(* CODESYS project CutToLength Prog final.project

Project tree, tasks and I/O mapping:
  Drive : Unidrive M701, Nidec Control Techniques, version 1.10.1.9
    application Application
      Program/
        program Freewheeling [LD]
      Codesys Setup/
        libraries: CT Unidrive M Parameter Library, * (Control Techniques); CT Unidrive M Options Parameter Library, 1.10.1.9 (Control Techniques)
        Task Configuration
          Freewheeling
      Basic AMC Library/
        03 Commands/
          Stop/
            function Stop_Motion [ST]
            function Stop_Motion_Decel [ST]
          Home/
            function Set_Position [ST]
            function Start_Homing_To_Input_4 [ST]
            function Start_Homing_To_Input_4_Then_Marker [ST]
            function Start_Homing_To_Torque [ST]
            function Start_Homing_To_Torque_Then_Input_4 [ST]
            function Start_Homing_To_Torque_Then_Marker [ST]
          Jog/
            function Start_Jog_Minus [ST]
            function Start_Jog_Plus [ST]
          Index/
            function Start_Index_ABS [ST]
            function Start_Index_INC [ST]
            function Start_Index_REF [ST]
          EGB/
            function Start_Gearing [ST]
        01 Setup/
          function AMC_Enable [ST]
          function AMC_MasterUnits [ST]
          function AMC_UserUnits [ST]
          function AMC_StopMode [ST]
        10 Other/
          function ScaleValue_DI [ST]
          function Wait_Time [ST]
        02 Feedback/
      Variables/
        AMC Variables/
          global variables gvAMC_Flags
          global variables gvAMC_Windows
          global variables gvAMC_SoftPosLimit
          global variables gvAMC_Profile
          global variables gvAMC_HardPosLimit
          global variables gvAMC_Positions
          global variables gvAMC_Cam
          global variables gvAMC_Speed
        M701 DRIVE /
          global variables gvDrive_Commands
          global variables gvDrive_Limits
          global variables gvDrive_Flags
          global variables gvDrive_Analog
          global variables gvDrive_Digital_States
          global variables gvDrive_Info
          global variables gvDrive_Keypad
          global variables gvDrive_PID1
          global variables gvDrive_PID2
          global variables gvDrive_Menu18
          global variables gvDrive_Menu19
          global variables gvDrive_Menu20
          global variables gvDrive_Digital_Inverts
        data type eMotionID
    <Empty>
    <Empty>
    <Empty>
  Advanced Link Editor
    DefaultSection
*)

// Drive/Application/Variables/eMotionID
//This enum can be used to identify the motion.

{attribute 'qualified_only'}
TYPE eMotionID :
(
	
	NA :=0,
	AbsIndex_001 		:=101,
	AbsIndex_002 		:=102,
	AbsIndex_003 		:=103,
	AbsIndex_004 		:=104,
	AbsIndex_005 		:=105,
	AbsIndex_006 		:=106,
	AbsIndex_007 		:=107,
	AbsIndex_008 		:=108,
	AbsIndex_009 		:=109,
	AbsIndex_010 		:=110, 
	
	RefIndex_001 		:=201,
	RefIndex_002 		:=202,
	RefIndex_003 		:=203,
	RefIndex_004 		:=204,
	RefIndex_005 		:=205,
	RefIndex_006 		:=206,
	RefIndex_007 		:=207,
	RefIndex_008 		:=208,
	RefIndex_009 		:=209,
	RefIndex_010 		:=210, 
	
	IncIndex_001 		:=301,
	IncIndex_002 		:=302,
	IncIndex_003 		:=303,
	IncIndex_004 		:=304,
	IncIndex_005 		:=305,
	IncIndex_006 		:=306,
	IncIndex_007 		:=307,
	IncIndex_008 		:=308,
	IncIndex_009 		:=309,
	IncIndex_010 		:=310,  

	JogPlus_001			:=401,
	JogPlus_002			:=402,
	JogPlus_003			:=403,
	JogPlus_004			:=404,
	JogPlus_005			:=405,
	JogPlus_006			:=406,
	JogPlus_007			:=407,
	JogPlus_008			:=408,
	JogPlus_009			:=409,
	JogPlus_010			:=410,

	JogMinus_001		:=501,
	JogMinus_002		:=502,
	JogMinus_003		:=503,
	JogMinus_004		:=504,
	JogMinus_005		:=505,
	JogMinus_006		:=506,
	JogMinus_007		:=507,
	JogMinus_008		:=508,
	JogMinus_009		:=509,
	JogMinus_010		:=510,

	Gearing_001			:=601,
	Gearing_002			:=602,
	Gearing_003			:=603,
	Gearing_004			:=604,
	Gearing_005			:=605,
	Gearing_006			:=606,
	Gearing_007			:=607,
	Gearing_008			:=608,
	Gearing_009			:=609,
	Gearing_010			:=610,

	Cam_001				:=701,
	Cam_002				:=702,
	Cam_003				:=703,
	Cam_004				:=704,
	Cam_005				:=705,
	Cam_006				:=706,
	Cam_007				:=707,
	Cam_008				:=708,
	Cam_009				:=709,
	Cam_010				:=710,

	Home_001			:=801,
	Home_002			:=802,
	Home_003			:=803,
	Home_004			:=804,
	Home_005			:=805,
	Home_006			:=806,
	Home_007			:=807,
	Home_008			:=808,
	Home_009			:=809,
	Home_010			:=810,
	
	
	Error	 := -1		 //
)INT;
END_TYPE

// Drive/Application/Variables/AMC Variables/gvAMC_Flags
{attribute 'qualified_only'}
VAR_GLOBAL
	
 	//(33.010) [Get:Set] AMC Slave Freeze Flag, 
	//Slave freeze flag status parameter 33.010. 
	{attribute 'get_access' := 'ReadUserParameterBOOL(00,33,010)'}
	{attribute 'set_access' := 'WriteUserParameterBOOL(00,33,010,CaptureFlag_1)'}
	{attribute 'monitoring_instead' := 'ReadUserParameterBOOL(00,33,010)'}
	CaptureFlag_1: BOOL;

	
	//(32.010) [Get:Set] AMC Master Freeze Flag, 
	//Master freeze flag status.  
	{attribute 'get_access' := 'ReadUserParameterBOOL(00,32,010)'}
	{attribute 'set_access' := 'WriteUserParameterBOOL(00,32,010,CaptureFlag_2)'}
	{attribute 'monitoring_instead' := 'ReadUserParameterBOOL(00,32,010)'}
	CaptureFlag_2: BOOL;

	
	//(37.006) AMC EGB Locked,[Get] , 
	//Displays when the electronic gearbox is locked.  
	{attribute 'get_access' := 'ReadUserParameterBOOL(00,37,006)'}
	{attribute 'monitoring_instead' := 'ReadUserParameterBOOL(00,37,006)'}
	EGB_Locked: BOOL;
	

	//(41.004) AMC Movement Complete Flag[Get] 
	//range 0 to 1 - precision is 0 decimal places.
	//NOTE:  There is a 4ms update delay for this Parameter. 
	{attribute 'get_access' := 'ReadUserParameterBOOL(00,41,004)'}
	{attribute 'monitoring_instead' := 'ReadUserParameterBOOL(00,41,004)'}
	MovementCompleteFlag: BOOL;
	
	
	//(41.004) AMC Profile Complete Flag[Get] 
	//range 0 to 1 - precision is 0 decimal places.
	//NOTE:  There is a 4ms update delay for this Parameter. 
	{attribute 'get_access' := 'ReadUserParameterBOOL(00,41,006)'}
	{attribute 'monitoring_instead' := 'ReadUserParameterBOOL(00,41,006)'}
	ProfileCompleteFlag: BOOL;
	
	
	//(40.005)[Get] Home Complete Flag 
	//Indiates that the Home is Complete.  If the Home has a offset position command the motor 
	//might not be done moving to the offset position.
	{attribute 'get_access' := 'ReadUserParameterBOOL(00,40,005)'}
	{attribute 'monitoring_instead' := 'ReadUserParameterBOOL(00,40,005)'}
	HomeCompleteFlag : BOOL;
	
		
	//(40.007)[Get] Home Complete with Offset Complete
	//Indiates that the Home and the offset move is Complete.  If the Home has a offset position command the motor 
	//might not be done moving to the offset position.
	{attribute 'get_access' := 'ReadUserParameterBOOL(00,40,008)'}
	{attribute 'monitoring_instead' := 'ReadUserParameterBOOL(00,40,008)'}
	HomeOffsetCompleteFlag : BOOL;
	 
	
	//(41.008)[Get] AMC Following Error Flag 
	//Indiates that the position error is outside the follwing error window Parameter 41.007
	{attribute 'get_access' := 'ReadUserParameterBOOL(00,41,008)'}
	{attribute 'monitoring_instead' := 'ReadUserParameterBOOL(00,41,008)'}
	FollowingErrorFlag : BOOL;
	 
	//(41.010)[Get] AMC Speed Error Flag 
	//Indiates that the position error is outside the follwing error window Parameter 41.010
	{attribute 'get_access' := 'ReadUserParameterBOOL(00,41,010)'}
	{attribute 'monitoring_instead' := 'ReadUserParameterBOOL(00,41,010)'}
	SpeedErrorFlag : BOOL;
	 
	//(41.012) [Get] AMC Following Error Stop Flag 
	{attribute 'get_access' := 'ReadUserParameterBOOL(00,41,012)'}
	{attribute 'monitoring_instead' := 'ReadUserParameterBOOL(00,41,012)'}
	FollowingErrorStop: BOOL;

	//(41.013)[Get] AMC Positive Hardware Limit Flag 
	{attribute 'get_access' := 'ReadUserParameterBOOL(00,41,013)'}
	{attribute 'monitoring_instead' := 'ReadUserParameterBOOL(00,41,013)'}
	Positive_HardwareLimit: BOOL;
	
	//(41.014) [Get] AMC Negative Hardware Limit Flag 
	{attribute 'get_access' := 'ReadUserParameterBOOL(00,41,014)'}
	{attribute 'monitoring_instead' := 'ReadUserParameterBOOL(00,41,014)'}
	Negative_HardwareLimit: BOOL;
	
	//(41.015) [Get] AMC Positive Software Limit Flag 
	{attribute 'get_access' := 'ReadUserParameterBOOL(00,41,015)'}
	{attribute 'monitoring_instead' := 'ReadUserParameterBOOL(00,41,015)'}
	Positive_SoftwareLimit: BOOL;
	
	//(41.016) [Get] AMC Negative Software Limit Flag 
	{attribute 'get_access' := 'ReadUserParameterBOOL(00,41,016)'}
	{attribute 'monitoring_instead' := 'ReadUserParameterBOOL(00,41,016)'}
	Negative_SoftwareLimit: BOOL;
	
	//(41.017)[Get] AMC Home Required Flag, 
	{attribute 'get_access' := 'ReadUserParameterBOOL(00,41,017)'}
	{attribute 'monitoring_instead' := 'ReadUserParameterBOOL(00,41,017)'}
	HomeRequired: BOOL;
	
	
	
END_VAR

// Drive/Application/Variables/AMC Variables/gvAMC_Windows
{attribute 'qualified_only'}
VAR_GLOBAL
	

	//(41.003) AMC Movement Complete Window [Get:Set] 
	// range -2147483648 to 2147483647UU - precision is 0 decimal places.
	{attribute 'get_access' 		:= 'ReadUserParameterDINT(00,41,003)'}
	{attribute 'set_access' 		:= 'WriteUserParameterDINT(00,41,003,MovementCompleteWindow)'}
	{attribute 'monitoring_instead' := 'ReadUserParameterDINT(00,41,003)'}
	MovementCompleteWindow: DINT; 

	//(41.005) AMC Profile Complete Window [Get:Set] 
	// range -2147483648 to 2147483647UU - precision is 0 decimal places.
	{attribute 'get_access' 		:= 'ReadUserParameterDINT(00,41,005)'}
	{attribute 'set_access' 		:= 'WriteUserParameterDINT(00,41,005,ProfileCompleteWindow)'}
	{attribute 'monitoring_instead' := 'ReadUserParameterDINT(00,41,005)'}
	ProfileCompleteWindow: DINT; 

	//(41.007) AMC Following Error Window [Get:Set] 
	// range -2147483648 to 2147483647UU - precision is 0 decimal places.
	{attribute 'get_access' 		:= 'ReadUserParameterDINT(00,41,007)'}
	{attribute 'set_access' 		:= 'WriteUserParameterDINT(00,41,007,FollowingErrorWindow)'}
	{attribute 'monitoring_instead' := 'ReadUserParameterDINT(00,41,007)'}
	FollowingErrorWindow: DINT; 

	//(41.009) AMC At Speed Window [Get:Set] 
	// range -2147483648 to 2147483647UU - precision is 0 decimal places.
	{attribute 'get_access' 		:= 'ReadUserParameterDINT(00,41,009)'}
	{attribute 'set_access' 		:= 'WriteUserParameterDINT(00,41,009,AtSpeedWindow)'}
	{attribute 'monitoring_instead' := 'ReadUserParameterDINT(00,41,009)'}
	AtSpeedWindow: DINT; 
	
	
	
END_VAR

// Drive/Application/Variables/AMC Variables/gvAMC_SoftPosLimit
{attribute 'qualified_only'}
VAR_GLOBAL
  
	
 	//(41.024) AMC Enable Software Limits, [Get:Set], 
	//range 0 to 1   
	//Value of 0 = Profile
	//Value of 1 = No Profile
	{attribute 'get_access' 		:= 'ReadUserParameterSINT (00,41,024)'}
	{attribute 'set_access' 		:= 'WriteUserParameterSINT(00,41,024,SoftwareLimitStopMode)'}
	{attribute 'monitoring_instead' := 'ReadUserParameterSINT (00,41,024)'}
	SoftwareLimitStopMode		: SINT;
	 
  	//(41.025) AMC Enable Software Limits, [Get:Set], 
	//range 0 to 1   
	{attribute 'get_access' 		:= 'ReadUserParameterBOOL (00,41,025)'}
	{attribute 'set_access' 		:= 'WriteUserParameterBOOL(00,41,025,EnableSoftwareLimits)'}
	{attribute 'monitoring_instead' := 'ReadUserParameterBOOL (00,41,025)'}
	EnableSoftwareLimits		: BOOL;	 
	
	//(41.026)AMC Positive Software Limit Position, [Get:Set] , 
	//range -2147483648 to 2147483647UU - precision is 0 decimal places. 
	{attribute 'get_access' 		:= 'ReadUserParameterDINT  (00,41,026)'}
	{attribute 'set_access' 		:= 'WriteUserParameterDINT (00,41,026,PositiveSoftwareLimitPosition)'}
	{attribute 'monitoring_instead' := 'ReadUserParameterDINT  (00,41,026)'}
	PositiveSoftwareLimitPosition: DINT;
	
	
	//(41.027) AMC Negative Software Limit Position, [Get:Set] , 
	//range -2147483648 to 2147483647UU - precision is 0 decimal places. 
	{attribute 'get_access' 		:= 'ReadUserParameterDINT (00,41,027)'}
	{attribute 'set_access' 		:= 'WriteUserParameterDINT(00,41,027,NegativeSoftwareLimitPosition)'}
	{attribute 'monitoring_instead' := 'ReadUserParameterDINT (00,41,027)'}
	NegativeSoftwareLimitPosition: DINT;
	
	
	
END_VAR

// Drive/Application/Variables/AMC Variables/gvAMC_Profile
{attribute 'qualified_only'}
VAR_GLOBAL
	
  
	
	//(38.001) [Get:Set] AMC Profile Acceleration, range -2147483648 to 2147483647UU/ms²
	// precision is 3 decimal places.
	// Unit are in User units / ms² 
	{attribute 'get_access' 		:= 'ReadUserParameterDINT(00,38,001)'}
	{attribute 'set_access' 		:= 'WriteUserParameterDINT(00,38,001,Acceleration)'}
	{attribute 'monitoring_instead' := 'ReadUserParameterDINT(00,38,001)'}
	Acceleration: DINT; 
	
	//(38.002) [Get:Set] AMC Profile Deceleration, range -2147483648 to 2147483647UU/ms²
	// precision is 3 decimal places.
	// Unit are in User units / ms² 
	{attribute 'get_access' 		:= 'ReadUserParameterDINT(00,38,002)'}
	{attribute 'set_access' 		:= 'WriteUserParameterDINT(00,38,002,Deceleration)'}
	{attribute 'monitoring_instead' := 'ReadUserParameterDINT(00,38,002)'}
	Deceleration: DINT; 
	
	//(38.003) [Get:Set] AMC Profile Maximum Speed, range -2147483648 to 2147483647UU/ms
	//precision is 2 decimal places.
	//Unit are in User units / ms
	{attribute 'get_access' 		:= 'ReadUserParameterDINT(00,38,003)'}
	{attribute 'set_access' 		:= 'WriteUserParameterDINT(00,38,003,MaximumSpeed)'}
	{attribute 'monitoring_instead' := 'ReadUserParameterDINT(00,38,003)'}
	MaximumSpeed: DINT;
	
	
END_VAR

// Drive/Application/Variables/AMC Variables/gvAMC_HardPosLimit
{attribute 'qualified_only'}
VAR_GLOBAL
	 

	//(41.023) AMC Hardware Limit Stop Mode, [Get:Set]  
	//Stop mode used when a hardware limit are active. 
	//Value of 0 = Profile
	//Value of 1 = No Profile
	//This uses parameter 6.035 and parameter 6.036.
	//parameter 06.035 is Forward Limit Switch 
	//parameter 06.036 is Reverse Limit Switch
	//These two parameters are controled by anything you map to it.  Most of the time a digital input will control them.
	//Example:  Set parameter 8.025 = 6.035 and set parameter 8.026 = 6.036.  Now digital input 5 and 6 control the hardware limits.
	{attribute 'get_access' 		:= 'ReadUserParameterSINT(00,41,023)'}
	{attribute 'set_access' 		:= 'WriteUserParameterSINT(00,41,023,HardwareLimitSwitch_NoRamp_StopMode)'}
	{attribute 'monitoring_instead' := 'ReadUserParameterSINT(00,41,023)'}	
	HardwareLimitSwitch_NoRamp_StopMode			: SINT;
 
   
	 
	 
	
END_VAR

// Drive/Application/Variables/AMC Variables/gvAMC_Positions
{attribute 'qualified_only'}
VAR_GLOBAL
	 

	//(33.004) [Get] System Position, range -2147483648 to 2147483647UU - 
	//precision is 0 decimal places.
	//Displays the AMC Slave Position. 
	//Update Rate 4ms
	{attribute 'get_access' 		:= 'ReadUserParameterDINT(00,33,004)'}
	{attribute 'monitoring_instead' := 'ReadUserParameterDINT(00,33,004)'}
	SystemPosition: DINT;
  
  	//(32.004) [Get] Master Position, range -2147483648 to 2147483647UU -
	//precision is 0 decimal places. 
	//Displays the AMC Slave Position. 
	//Update Rate 4ms
	{attribute 'get_access' 		:= 'ReadUserParameterDINT(00,32,004)'}
	{attribute 'monitoring_instead' := 'ReadUserParameterDINT(00,32,004)'}
	MasterPosition: DINT; 
	
	 
	//[Get] AMC Slave Freeze Position(33.006),  
	//Displays the AMC Slave Position after a freeze event has occurred. 
	{attribute 'get_access' 		:= 'ReadUserParameterDINT(00,33,006)'}
	{attribute 'monitoring_instead' := 'ReadUserParameterDINT(00,33,006)'}
	CapturedPosition_1: DINT;
	
	
	///[Get] AMC Master Freeze Position(32.006), 
	//Displays the AMC Slave Position after a freeze event has occurred. 
	{attribute 'get_access' 		:= 'ReadUserParameterDINT(00,32,006)'}
	{attribute 'monitoring_instead' := 'ReadUserParameterDINT(00,32,006)'}
	CapturedPosition_2: DINT;
	
	
END_VAR

// Drive/Application/Variables/M701 DRIVE /gvDrive_Commands
{attribute 'qualified_only'}
VAR_GLOBAL
	 

	//(06.008)Hold Zero Speed [Get:Set] 
	//If True then the drive will hold a zero speed command even if no run command is given
	{attribute 'get_access' 		:= 'ReadUserParameterBOOL (00,06,008)'}
	{attribute 'set_access' 		:= 'WriteUserParameterBOOL(00,06,008,HoldZeroSpeed)'}
	{attribute 'monitoring_instead' := 'ReadUserParameterBOOL (00,06,008)'}
	HoldZeroSpeed : BOOL;

	
	//(06.030) Basic Run Forward [Get:Set] 
	//Needs to be true before anymoon commands will operate.
	{attribute 'get_access' 		:= 'ReadUserParameterBOOL (00,06,030)'}
	{attribute 'set_access' 		:= 'WriteUserParameterBOOL(00,06,030,RunForward)'}
	{attribute 'monitoring_instead' := 'ReadUserParameterBOOL (00,06,030)'}
	RunForward: BOOL;
	
	 
	//(06.032) Basic Run Reverse [Get:Set] 
	//Needs to be true before anymoon commands will operate.
	{attribute 'get_access' 		:= 'ReadUserParameterBOOL (00,06,032)'}
	{attribute 'set_access' 		:= 'WriteUserParameterBOOL(00,06,032,RunReverse)'}
	{attribute 'monitoring_instead' := 'ReadUserParameterBOOL (00,06,032)'}
	RunReverse: BOOL;
	
	
	
END_VAR

// Drive/Application/Variables/M701 DRIVE /gvDrive_Limits
{attribute 'qualified_only'}
VAR_GLOBAL
	

 
	//(04.005) Motoring Current Limit [Get:Set], range 0.0 to 1000.0%
	//Defines the current limit used when the motor is being accelerated away from standstill. 
	{attribute 'get_access' 		:= 'ReadUserParameterINT (00,04,005)'}
	{attribute 'set_access' 		:= 'WriteUserParameterINT(00,04,005,MotorCurrentLimit_RAW)'}
	{attribute 'monitoring_instead' := 'ReadUserParameterINT (00,04,005)'}
	MotorCurrentLimit_RAW: INT;
 
	
	//(04.006) Regenerating Current Limit [Get:Set], range 0.0 to 1000.0%
	//Defines the current limit used when the motor is being decelerated towards standstill. 
	{attribute 'get_access' 		:= 'ReadUserParameterINT (00,04,006)'}
	{attribute 'set_access' 		:= 'WriteUserParameterINT(00,04,006,RegCurrentLimit_RAW)'}
	{attribute 'monitoring_instead' := 'ReadUserParameterINT (00,04,006)'}
	RegCurrentLimit_RAW: INT;  
	
 
	//(03.008) Over Speed Threshold, range 0.0 to 3000.0Hz
	//Set to the required over speed threshold. 
	{attribute 'get_access' 		:= 'ReadUserParameterUINT(00,03,008)'}
	{attribute 'set_access'	 		:= 'WriteUserParameterUINT(00,03,008,OverSpeedThreshold_RAW)'}
	{attribute 'monitoring_instead' := 'ReadUserParameterUINT(00,03,008)'}
	OverSpeedThreshold_RAW: UINT; 
	
	
	//(01.006) Maximum Reference Clamp [Get:Set], range -2147483648 to 2147483647 - precision is 1 decimal places.
	//Defines the maximum value for the reference. 
	{attribute 'get_access' 		:= 'ReadUserParameterDINT(00,01,006)'}
	{attribute 'set_access' 		:= 'WriteUserParameterDINT(00,01,006,MaximumReferenceClamp_RAW)'}
	{attribute 'monitoring_instead' := 'ReadUserParameterDINT(00,01,006)'}
	MaximumReferenceClamp_RAW: DINT; 
	
	
	//(01.007) Minimum Reference Clamp [Get:Set], range -2147483648 to 2147483647 - precision is 1 decimal places.
	//Defines the minimum value for the reference.  
	{attribute 'get_access' 		:= 'ReadUserParameterDINT(00,01,007)'}
	{attribute 'set_access' 		:= 'WriteUserParameterDINT(00,01,007,MinimumReferenceClamp_RAW)'}
	{attribute 'monitoring_instead' := 'ReadUserParameterDINT(00,01,007)'}
	MinimumReferenceClamp_RAW: DINT;

	
END_VAR

// Drive/Application/Variables/M701 DRIVE /gvDrive_Flags
{attribute 'qualified_only'}
VAR_GLOBAL
	
	//(10.001)[Get] Drive Healthy,  
	//Indicates that the drive is healthy. 
	{attribute 'get_access' 		:= 'ReadUserParameterBOOL(00,10,001)'}
	{attribute 'monitoring_instead' := 'ReadUserParameterBOOL(00,10,001)'}
	DriveHealthy: BOOL;
	
	//(10.003)[Get] Zero Speed,  
	//Indicates that the speed is below the zero speed threshold. 
	//Zero Speed is set to TRUE, IF the Speed Feedback parameter (03.002) 
	//is AT OR below Zero Speed Threshold (03.005).  
	{attribute 'get_access' 		:= 'ReadUserParameterBOOL(00,10,003)'}
	{attribute 'monitoring_instead' := 'ReadUserParameterBOOL(00,10,003)'}
	ZeroSpeed: BOOL;
	
	//(10.006)[Get] At Speed 
	//Indicates that the drive is running at the set speed.  
	//At Speed (10.006) is set if the Speed Feedback (03.002) is on the boundaries or 
	//within the at speed window. Above Set Speed (10.007) and Below Set Speed (10.005) 
	//are set if the feedback is above or below the window respectively.
	{attribute 'get_access' 		:= 'ReadUserParameterBOOL(00,10,006)'}
	{attribute 'monitoring_instead' := 'ReadUserParameterBOOL(00,10,006)'}
	AtSpeed : BOOL;
	
	//(10.009)[Get] Current Limit Active,  
	//Indicates that the current limit is active.  
	//is set to one if the current limit is active. 
	//It should be noted that the current limit system is used in RFC-A and RFC-S modes 
	//when standard ramp control is active (Ramp Mode (02.004)), or supply loss control 
	//is in ramp stop or limit stop mode (Supply Loss Mode (06.003)). 
	//Therefore Current Limit Active (10.009) is likely to change to one under these 
	//conditions, even if the user defined current limits are not active.
	{attribute 'get_access' 		:= 'ReadUserParameterBOOL(00,10,009)'}
	{attribute 'monitoring_instead' := 'ReadUserParameterBOOL(00,10,009)'}
	CurrentLimitActive: BOOL;

  	//(10.014)[Get] Reverse Direction Running 
	//Indicates that the drive is running in the reverse direction.  
	//Is set to one if the Speed Feedback (03.002) is negative otherwise it is set to zero. 
	{attribute 'get_access' 		:= 'ReadUserParameterBOOL(00,10,014)'}
	{attribute 'monitoring_instead' := 'ReadUserParameterBOOL(00,10,014)'}
	ReverseDirectionRunning : BOOL;
	
	
END_VAR

// Drive/Application/Variables/M701 DRIVE /gvDrive_Analog
{attribute 'qualified_only'}
VAR_GLOBAL
	
	// 07.001
   	// Analog Input 1(07.001), range -100.00-100.00
    {attribute 'get_access' 		:= 'ReadUserParameterINT(00,07,001)'}
    {attribute 'monitoring_instead' := 'ReadUserParameterINT(00,07,001)'}
    Input1_RAW : INT; 

	// 07.002
    // Analog Input 2(07.002), range -100.00-100.00.
    {attribute 'get_access' 		:= 'ReadUserParameterINT(00,07,002)'}
    {attribute 'monitoring_instead' := 'ReadUserParameterINT(00,07,002)'}
    Input2_RAW : INT;


	// 07.003
    // Analog Input 3(07.003), range -100.00-100.00.
    {attribute 'get_access' 		:= 'ReadUserParameterINT(00,07,003)'}
    {attribute 'monitoring_instead' := 'ReadUserParameterINT(00,07,003)'}
    Input3_RAW : INT;



END_VAR

// Drive/Application/Variables/M701 DRIVE /gvDrive_Digital_States
(*
	If you change the name of the inverts in this list you also have to change the set_access line of code.
	
*)

{attribute 'qualified_only'}
VAR_GLOBAL
	
	// M08.P001
    // Digital I/O 01 State
    {attribute 'get_access' 		:= 'ReadUserParameterBOOL(00,08,001)'}
    {attribute 'monitoring_instead' := 'ReadUserParameterBOOL(00,08,001)'}
    IO_01 : BOOL;

	// M08.P002	
    // Digital I/O 02 State 
    {attribute 'get_access' 		:= 'ReadUserParameterBOOL(00,08,002)'}
    {attribute 'monitoring_instead' := 'ReadUserParameterBOOL(00,08,002)'}
    IO_02 : BOOL;

	// M08.P003
    // Digital I/O 03 State 
    {attribute 'get_access' 		:= 'ReadUserParameterBOOL(00,08,003)'}
    {attribute 'monitoring_instead' := 'ReadUserParameterBOOL(00,08,003)'}
    IO_03: BOOL;

	// M08.P004
    // Digital Input 04 State 
    {attribute 'get_access' 		:= 'ReadUserParameterBOOL(00,08,004)'}
    {attribute 'monitoring_instead' := 'ReadUserParameterBOOL(00,08,004)'}
    Input04 : BOOL;
	
	// M08.P005
    // Digital Input 05 State
    {attribute 'get_access' 		:= 'ReadUserParameterBOOL(00,08,005)'}
    {attribute 'monitoring_instead' := 'ReadUserParameterBOOL(00,08,005)'}
    Input05: BOOL;

	// M08.P006
    // Digital Input 06 State
    {attribute 'get_access' 		:= 'ReadUserParameterBOOL(00,08,006)'}
    {attribute 'monitoring_instead' := 'ReadUserParameterBOOL(00,08,006)'}
    Input06 : BOOL;
 
	// M08.P007
    // Relay Output State 
    {attribute 'get_access' 		:= 'ReadUserParameterBOOL(00,08,007)'}
    {attribute 'monitoring_instead' := 'ReadUserParameterBOOL(00,08,007)'}
    RelayOutput07 : BOOL;

	// M08.P008
    // 24V Supply Output State 
    {attribute 'get_access' 		:= 'ReadUserParameterBOOL(00,08,008)'}
    {attribute 'monitoring_instead' := 'ReadUserParameterBOOL(00,08,008)'}
    VoltageSupplyOutputState  		: BOOL;

	// M08.P043
    // 24V Supply Input State 
	// Turns on when the drive is given 24v from a power supply 
    {attribute 'get_access' 		:= 'ReadUserParameterBOOL(00,08,008)'}
    {attribute 'monitoring_instead' := 'ReadUserParameterBOOL(00,08,008)'}
    VoltageSupplyInputState  		: BOOL;

	// M08.P009
    // STO Input 01 State
    {attribute 'get_access' 		:= 'ReadUserParameterBOOL(00,08,009)'}
    {attribute 'monitoring_instead' := 'ReadUserParameterBOOL(00,08,009)'}
    SaftTorqueOff1 : BOOL;

	// M08.P040	
	// STO Input 02 State 
    {attribute 'get_access' 		:= 'ReadUserParameterBOOL(00,08,040)'}
    {attribute 'monitoring_instead' := 'ReadUserParameterBOOL(00,08,040)'}
    SaftTorqueOff2 : BOOL;

END_VAR

// Drive/Application/Variables/M701 DRIVE /gvDrive_Info
{attribute 'qualified_only'}
VAR_GLOBAL
	

	//(03.002) Speed Feedback, 1 decimal places.
	//Displays the speed feedback from the selected feedback source. 
	{attribute 'get_access' 		:= 'ReadUserParameterLREAL(00,03,002)'}
	{attribute 'monitoring_instead' := 'ReadUserParameterLREAL(00,03,002)'}
	SpeedFeedback: LREAL;
	
	//(03.002) Speed Feedback, 1 decimal place, Value of 1000 = 100.0 RPM
	///Displays the speed feedback from the selected feedback source. 
	{attribute 'get_access' 		:= 'ReadUserParameterDINT(00,03,002)'}
	{attribute 'monitoring_instead' := 'ReadUserParameterDINT(00,03,002)'}
	SpeedFeedback_RAW: DINT;	
	
	//(04.001) Current Magnitude, 3 decimal places.
	//Shows the instantaneous drive output current.  
	{attribute 'get_access' 		:= 'ReadUserParameterLREAL(00,04,001)'}
	{attribute 'monitoring_instead' := 'ReadUserParameterLREAL(00,04,001)'}
	CurrentMagnitude: LREAL;	
	
	//(04.001) Current Magnitude, 3 decimal places, Value of 1000 = 1.000amps
	//Shows the instantaneous drive output current.  
	{attribute 'get_access' 		:= 'ReadUserParameterDINT(00,04,001)'}
	{attribute 'monitoring_instead' := 'ReadUserParameterDINT(00,04,001)'}
	CurrentMagnitude_RAW: DINT;	
	
	//(06.043) Control Word Enable,  
	//Set to 1 to enable the control word. - All Modes
	//if on then the control word is used to give the drive run commands
	{attribute 'get_access' 		:= 'ReadUserParameterBOOL(00,06,043)'} 
	{attribute 'set_access' 		:= 'WriteUserParameterBOOL(00,06,043,ControlWordEnable)'}
	{attribute 'monitoring_instead' := 'ReadUserParameterBOOL(00,06,043)'}
	ControlWordEnable: BOOL;
	
END_VAR

// Drive/Application/Variables/M701 DRIVE /gvDrive_Keypad
{attribute 'qualified_only'}
VAR_GLOBAL
	
 
	// M08.P041	Run Button
    {attribute 'get_access' 		:= 'ReadUserParameterBOOL(00,08,041)'}
    {attribute 'monitoring_instead' := 'ReadUserParameterBOOL(00,08,041)'}
    RunButton : BOOL;

	// M08.P042	Auxiliary Button
    {attribute 'get_access' 		:= 'ReadUserParameterBOOL(00,08,042)'}
    {attribute 'monitoring_instead' := 'ReadUserParameterBOOL(00,08,042)'}
    AuxiliaryButton : BOOL;

	// M08.P044	Auxiliary Button
    {attribute 'get_access' 		:= 'ReadUserParameterBOOL(00,08,044)'}
    {attribute 'monitoring_instead' := 'ReadUserParameterBOOL(00,08,044)'}
    StopButton : BOOL;


END_VAR

// Drive/Application/Variables/M701 DRIVE /gvDrive_PID1
(*
	See menu 14 for all of th PID settings.
*)
{attribute 'qualified_only'}
VAR_GLOBAL
		
	//(14.008) [Get:Set] PID1 Enable, 
	//Enables the use of PID1
	//Note there are also two other parameters they can be used to encable the PID
	//Parameter 14.009 and parameter 14.027
	{attribute 'get_access' 		:= 'ReadUserParameterBOOL(00,14,008)'}
	{attribute 'set_access' 		:= 'WriteUserParameterBOOL(00,14,008,Enable)'}
	{attribute 'monitoring_instead' := 'ReadUserParameterBOOL(00,14,008)'}
	Enable: BOOL;
	
	//(14.001) [Get] PID1 Output, range -100.00 to 100.00%
	//Displays the output for PID1. 
	{abvibute 'get_access' 			:= 'ReadUserParameterINT(00,14,001)'}
	{attribute 'monitoring_instead' := 'ReadUserParameterINT(00,14,001)'}
	Output_RAW: INT;

	//(14.007) [Get:Set] PID1 Reference Slew Rate, range 0.0 to 3200.0s
	//Defines the rate in change of output for PID1. 
	{attribute 'get_access' 		:= 'ReadUserParameterINT(00,14,007)'}
	{attribute 'set_access' 		:= 'WriteUserParameterINT(00,14,007,SlewRate_RAW)'}
	{attribute 'monitoring_instead' := 'ReadUserParameterINT(00,14,007)'}
	SlewRate_RAW: INT;
 
	//(14.025) [Get:Set] PID1 Digital Reference, range -100.00 to 100.00%
	//Defines the value of the digital reference for PID1. 
	//Used if the PLC is setting the Reference else the parameter 14.003 should be used.
	{attribute 'get_access' 		:= 'ReadUserParameterINT(00,14,025)'}
	{attribute 'set_access' 		:= 'WriteUserParameterINT(00,14,025,Reference_RAW)'}
	{attribute 'monitoring_instead' := 'ReadUserParameterINT(00,14,025)'}
	Reference_RAW: INT;

	//(14.026) [Get:Set] PID1 Digital Feedback, range -100.00 to 100.00%
	//Defines the value of the digital feedback for PID1. 
	//Usd if the PLC is setting the Feedback else the parameter 14.004 should be used.
	{attribute 'get_access' 		:= 'ReadUserParameterINT(00,14,026)'}
	{attribute 'set_access' 		:= 'WriteUserParameterINT(00,14,026,Feedback_RAW)'}
	{attribute 'monitoring_instead' := 'ReadUserParameterINT(00,14,026)'}
	Feedback_RAW: INT;
END_VAR

// Drive/Application/Variables/M701 DRIVE /gvDrive_PID2
(*
	See menu 14 for all of th PID settings.
*)
{attribute 'qualified_only'}
VAR_GLOBAL
	
	//(14.038) [Get:Set] PID2 Enable, 
	//Enables the use of PID2
	//Note there are also two other parameters they can be used to encable the PID
	//Parameter 14.039 and parameter 14.057
	{attribute 'get_access' 		:= 'ReadUserParameterBOOL(00,14,038)'}
	{attribute 'set_access' 		:= 'WriteUserParameterBOOL(00,14,038,Enable)'}
	{attribute 'monitoring_instead' := 'ReadUserParameterBOOL(00,14,038)'}
	Enable: BOOL;

	//(14.031) [Get] PID2 Output, range -100.00 to 100.00%
	//Displays the output for PID1. 
	{attribute 'get_access' 		:= 'ReadUserParameterINT(00,14,031)'}
	{attribute 'monitoring_instead' := 'ReadUserParameterINT(00,14,031)'}
	Output_RAW: INT;

	//(14.037) [Get:Set] PID2 Reference Slew Rate, range 0.0 to 3200.0s
	//Defines the rate in change of output for PID1. 
	{attribute 'get_access' 		:= 'ReadUserParameterINT(00,14,037)'}
	{attribute 'set_access' 		:= 'WriteUserParameterINT(00,14,037,SlewRate_RAW)'}
	{attribute 'monitoring_instead' := 'ReadUserParameterINT(00,14,037)'}
	SlewRate_RAW: INT;
 
	//(14.055) [Get:Set] PID2 Digital Reference, range -100.00 to 100.00%
	//Defines the value of the digital reference for PID1. 
	//Used if the PLC is setting the Reference else the parameter 14.003 should be used.
	{attribute 'get_access' 		:= 'ReadUserParameterINT(00,14,055)'}
	{attribute 'set_access' 		:= 'WriteUserParameterINT(00,14,055,Reference_RAW)'}
	{attribute 'monitoring_instead' := 'ReadUserParameterINT(00,14,055)'}
	Reference_RAW: INT;

	//(14.056) [Get:Set] PID2 Digital Feedback, range -100.00 to 100.00%
	//Defines the value of the digital feedback for PID1. 
	//Usd if the PLC is setting the Feedback else the parameter 14.004 should be used.
	{attribute 'get_access' 		:= 'ReadUserParameterINT(00,14,056)'}
	{attribute 'set_access' 		:= 'WriteUserParameterINT(00,14,056,Feedback_RAW)'}
	{attribute 'monitoring_instead' := 'ReadUserParameterINT(00,14,056)'}
	Feedback_RAW: INT;
END_VAR

// Drive/Application/Variables/M701 DRIVE /gvDrive_Menu18
(*
	Menu 18
*)
(*	LEVEL 2 SUPPORT
	Only change the variable name after you know how.
	don't add extra white spaces inside the attribute.
*)
(*
	If you change the name of any of them in this list you also have to change the set_access line of code.
	
	Example:
	change P001 to P001_count
	Then you also need to change the attributes
 
	before
	
	{attribute 'get_bitaccess' := 'ReadUserParameterBit(00,18,001,BITNR)'}
	{attribute 'get_access' := 'ReadUserParameterINT(00,18,001)'}
	{attribute 'set_bitaccess' := 'WriteUserParameterBit(00,18,001,BITNR,P001)'}
	{attribute 'set_access' := 'WriteUserParameterINT(00,18,001,P001)'}
	{attribute 'monitoring_instead' := 'ReadUserParameterINT(00,18,001)'}
	P001: INT;
	
	after change 
	
	{attribute 'get_bitaccess' := 'ReadUserParameterBit(00,18,001,BITNR)'}
	{attribute 'get_access' := 'ReadUserParameterINT(00,18,001)'}
	{attribute 'set_bitaccess' := 'WriteUserParameterBit(00,18,001,BITNR,P001_count)'}
	{attribute 'set_access' := 'WriteUserParameterINT(00,18,001,P001_count)'}
	{attribute 'monitoring_instead' := 'ReadUserParameterINT(00,18,001)'}
	P001_count: INT;
	
*)
{attribute 'qualified_only'}
VAR_GLOBAL
 
	
	//(18.001)
	//save on power down
	{attribute 'get_bitaccess' := 'ReadUserParameterBit(00,18,001,BITNR)'}
	{attribute 'get_access' := 'ReadUserParameterINT(00,18,001)'}
	{attribute 'set_bitaccess' := 'WriteUserParameterBit(00,18,001,BITNR,Length_mm)'}
	{attribute 'set_access' := 'WriteUserParameterINT(00,18,001,Length_mm)'}
	{attribute 'monitoring_instead' := 'ReadUserParameterINT(00,18,001)'}
	Length_mm: INT;
	
	//(18.002) 
	{attribute 'get_bitaccess' := 'ReadUserParameterBit(00,18,002,BITNR)'}
	{attribute 'get_access' := 'ReadUserParameterINT(00,18,002)'}
	{attribute 'set_bitaccess' := 'WriteUserParameterBit(00,18,002,BITNR,View_Speed_Percent)'}
	{attribute 'set_access' := 'WriteUserParameterINT(00,18,002,View_Speed_Percent)'}
	{attribute 'monitoring_instead' := 'ReadUserParameterINT(00,18,002)'}
	View_Speed_Percent: INT;
	
	// (18.003) 
	{attribute 'get_bitaccess' := 'ReadUserParameterBit(00,18,003,BITNR)'}
	{attribute 'get_access' := 'ReadUserParameterINT(00,18,003)'}
	{attribute 'set_bitaccess' := 'WriteUserParameterBit(00,18,003,BITNR,Drive_Status)'}
	{attribute 'set_access' := 'WriteUserParameterINT(00,18,003,Drive_Status)'}
	{attribute 'monitoring_instead' := 'ReadUserParameterINT(00,18,003)'}
	Drive_Status: INT;
	
	//(18.004) 
	{attribute 'get_bitaccess' := 'ReadUserParameterBit(00,18,004,BITNR)'}
	{attribute 'get_access' := 'ReadUserParameterINT(00,18,004)'}
	{attribute 'set_bitaccess' := 'WriteUserParameterBit(00,18,004,BITNR,Count_Display)'}
	{attribute 'set_access' := 'WriteUserParameterINT(00,18,004,Count_Display)'}
	{attribute 'monitoring_instead' := 'ReadUserParameterINT(00,18,004)'}
	Count_Display: INT;
	
	//(18.005) 
	{attribute 'get_bitaccess' := 'ReadUserParameterBit(00,18,005,BITNR)'}
	{attribute 'get_access' := 'ReadUserParameterINT(00,18,005)'}
	{attribute 'set_bitaccess' := 'WriteUserParameterBit(00,18,005,BITNR,View_Distance_Per_Motor_Turn)'}
	{attribute 'set_access' := 'WriteUserParameterINT(00,18,005,View_Distance_Per_Motor_Turn)'}
	{attribute 'monitoring_instead' := 'ReadUserParameterINT(00,18,005)'}
	View_Distance_Per_Motor_Turn: INT;
	
	//(18.006) 
	{attribute 'get_bitaccess' := 'ReadUserParameterBit(00,18,006,BITNR)'}
	{attribute 'get_access' := 'ReadUserParameterINT(00,18,006)'}
	{attribute 'set_bitaccess' := 'WriteUserParameterBit(00,18,006,BITNR,View_Distance_Per_Encoder_Turn)'}
	{attribute 'set_access' := 'WriteUserParameterINT(00,18,006,View_Distance_Per_Encoder_Turn)'}
	{attribute 'monitoring_instead' := 'ReadUserParameterINT(00,18,006)'}
	View_Distance_Per_Encoder_Turn: INT;
	
	//(18.007) 
	{attribute 'get_bitaccess' := 'ReadUserParameterBit(00,18,007,BITNR)'}
	{attribute 'get_access' := 'ReadUserParameterINT(00,18,007)'}
	{attribute 'set_bitaccess' := 'WriteUserParameterBit(00,18,007,BITNR,View_Acceleration_Position)'}
	{attribute 'set_access' := 'WriteUserParameterINT(00,18,007,View_Acceleration_Position)'}
	{attribute 'monitoring_instead' := 'ReadUserParameterINT(00,18,007)'}
	View_Acceleration_Position: INT;
	
	//(18.008)
	{attribute 'get_bitaccess' := 'ReadUserParameterBit(00,18,008,BITNR)'}
	{attribute 'get_access' := 'ReadUserParameterINT(00,18,008)'}
	{attribute 'set_bitaccess' := 'WriteUserParameterBit(00,18,008,BITNR,View_Decceleration_Position)'}
	{attribute 'set_access' := 'WriteUserParameterINT(00,18,008,View_Decceleration_Position)'}
	{attribute 'monitoring_instead' := 'ReadUserParameterINT(00,18,008)'}
	View_Decceleration_Position: INT;
	
	//(18.009)
	{attribute 'get_bitaccess' := 'ReadUserParameterBit(00,18,009,BITNR)'}
	{attribute 'get_access' := 'ReadUserParameterINT(00,18,009)'}
	{attribute 'set_bitaccess' := 'WriteUserParameterBit(00,18,009,BITNR,View_Jog_Acceleration)'}
	{attribute 'set_access' := 'WriteUserParameterINT(00,18,009,View_Jog_Acceleration)'}
	{attribute 'monitoring_instead' := 'ReadUserParameterINT(00,18,009)'}
	View_Jog_Acceleration: INT;
	
	//(18.010) 
	{attribute 'get_bitaccess' := 'ReadUserParameterBit(00,18,010,BITNR)'}
	{attribute 'get_access' := 'ReadUserParameterINT(00,18,010)'}
	{attribute 'set_bitaccess' := 'WriteUserParameterBit(00,18,010,BITNR,View_Jog_Decceleration)'}
	{attribute 'set_access' := 'WriteUserParameterINT(00,18,010,View_Jog_Decceleration)'}
	{attribute 'monitoring_instead' := 'ReadUserParameterINT(00,18,010)'}
	View_Jog_Decceleration: INT;
	
	//(18.011) 
	{attribute 'get_bitaccess' := 'ReadUserParameterBit(00,18,011,BITNR)'}
	{attribute 'get_access' := 'ReadUserParameterINT(00,18,011)'}
	{attribute 'set_bitaccess' := 'WriteUserParameterBit(00,18,011,BITNR,View_Jog_Speed)'}
	{attribute 'set_access' := 'WriteUserParameterINT(00,18,011,View_Jog_Speed)'}
	{attribute 'monitoring_instead' := 'ReadUserParameterINT(00,18,011)'}
	View_Jog_Speed: INT;
	
	//(18.012) 
	{attribute 'get_bitaccess' := 'ReadUserParameterBit(00,18,012,BITNR)'}
	{attribute 'get_access' := 'ReadUserParameterINT(00,18,012)'}
	{attribute 'set_bitaccess' := 'WriteUserParameterBit(00,18,012,BITNR,Speed_Percent)'}
	{attribute 'set_access' := 'WriteUserParameterINT(00,18,012,Speed_Percent)'}
	{attribute 'monitoring_instead' := 'ReadUserParameterINT(00,18,012)'}
	Speed_Percent: INT := 150;
	
	//(18.013) 
	{attribute 'get_bitaccess' := 'ReadUserParameterBit(00,18,013,BITNR)'}
	{attribute 'get_access' := 'ReadUserParameterINT(00,18,013)'}
	{attribute 'set_bitaccess' := 'WriteUserParameterBit(00,18,013,BITNR,Count_Preset)'}
	{attribute 'set_access' := 'WriteUserParameterINT(00,18,013,Count_Preset)'}
	{attribute 'monitoring_instead' := 'ReadUserParameterINT(00,18,013)'}
	Count_Preset: INT := 0;
	
	//(18.014) 
	{attribute 'get_bitaccess' := 'ReadUserParameterBit(00,18,014,BITNR)'}
	{attribute 'get_access' := 'ReadUserParameterINT(00,18,014)'}
	{attribute 'set_bitaccess' := 'WriteUserParameterBit(00,18,014,BITNR,P014)'}
	{attribute 'set_access' := 'WriteUserParameterINT(00,18,014,P014)'}
	{attribute 'monitoring_instead' := 'ReadUserParameterINT(00,18,014)'}
	P014: INT;
	
	//(18.015)
	{attribute 'get_bitaccess' := 'ReadUserParameterBit(00,18,015,BITNR)'}
	{attribute 'get_access' := 'ReadUserParameterINT(00,18,015)'}
	{attribute 'set_bitaccess' := 'WriteUserParameterBit(00,18,015,BITNR,P015)'}
	{attribute 'set_access' := 'WriteUserParameterINT(00,18,015,P015)'}
	{attribute 'monitoring_instead' := 'ReadUserParameterINT(00,18,015)'}
	P015: INT;
	
	//(18.016)
	{attribute 'get_bitaccess' := 'ReadUserParameterBit(00,18,016,BITNR)'}
	{attribute 'get_access' := 'ReadUserParameterINT(00,18,016)'}
	{attribute 'set_bitaccess' := 'WriteUserParameterBit(00,18,016,BITNR,P016)'}
	{attribute 'set_access' := 'WriteUserParameterINT(00,18,016,P016)'}
	{attribute 'monitoring_instead' := 'ReadUserParameterINT(00,18,016)'}
	P016: INT;
	
	//(18.017)
	{attribute 'get_bitaccess' := 'ReadUserParameterBit(00,18,017,BITNR)'}
	{attribute 'get_access' := 'ReadUserParameterINT(00,18,017)'}
	{attribute 'set_bitaccess' := 'WriteUserParameterBit(00,18,017,BITNR,P017)'}
	{attribute 'set_access' := 'WriteUserParameterINT(00,18,017,P017)'}
	{attribute 'monitoring_instead' := 'ReadUserParameterINT(00,18,017)'}
	P017: INT;
	
	//(18.018)
	{attribute 'get_bitaccess' := 'ReadUserParameterBit(00,18,018,BITNR)'}
	{attribute 'get_access' := 'ReadUserParameterINT(00,18,018)'}
	{attribute 'set_bitaccess' := 'WriteUserParameterBit(00,18,018,BITNR,P018)'}
	{attribute 'set_access' := 'WriteUserParameterINT(00,18,018,P018)'}
	{attribute 'monitoring_instead' := 'ReadUserParameterINT(00,18,018)'}
	P018: INT;
	
	//(18.019) 
	{attribute 'get_bitaccess' := 'ReadUserParameterBit(00,18,019,BITNR)'}
	{attribute 'get_access' := 'ReadUserParameterINT(00,18,019)'}
	{attribute 'set_bitaccess' := 'WriteUserParameterBit(00,18,019,BITNR,P019)'}
	{attribute 'set_access' := 'WriteUserParameterINT(00,18,019,P019)'}
	{attribute 'monitoring_instead' := 'ReadUserParameterINT(00,18,019)'}
	P019: INT;
	
	//(18.020)
	{attribute 'get_bitaccess' := 'ReadUserParameterBit(00,18,020,BITNR)'}
	{attribute 'get_access' := 'ReadUserParameterINT(00,18,020)'}
	{attribute 'set_bitaccess' := 'WriteUserParameterBit(00,18,020,BITNR,P020)'}
	{attribute 'set_access' := 'WriteUserParameterINT(00,18,020,P020)'}
	{attribute 'monitoring_instead' := 'ReadUserParameterINT(00,18,020)'}
	P020: INT;
	
	//(18.021)
	{attribute 'get_bitaccess' := 'ReadUserParameterBit(00,18,021,BITNR)'}
	{attribute 'get_access' := 'ReadUserParameterINT(00,18,021)'}
	{attribute 'set_bitaccess' := 'WriteUserParameterBit(00,18,021,BITNR,P021)'}
	{attribute 'set_access' := 'WriteUserParameterINT(00,18,021,P021)'}
	{attribute 'monitoring_instead' := 'ReadUserParameterINT(00,18,021)'}
	P021: INT;
	
	//(18.022) 
	{attribute 'get_bitaccess' := 'ReadUserParameterBit(00,18,022,BITNR)'}
	{attribute 'get_access' := 'ReadUserParameterINT(00,18,022)'}
	{attribute 'set_bitaccess' := 'WriteUserParameterBit(00,18,022,BITNR,P022)'}
	{attribute 'set_access' := 'WriteUserParameterINT(00,18,022,P022)'}
	{attribute 'monitoring_instead' := 'ReadUserParameterINT(00,18,022)'}
	P022: INT;
	
	//(18.023) 
	{attribute 'get_bitaccess' := 'ReadUserParameterBit(00,18,023,BITNR)'}
	{attribute 'get_access' := 'ReadUserParameterINT(00,18,023)'}
	{attribute 'set_bitaccess' := 'WriteUserParameterBit(00,18,023,BITNR,P023)'}
	{attribute 'set_access' := 'WriteUserParameterINT(00,18,023,P023)'}
	{attribute 'monitoring_instead' := 'ReadUserParameterINT(00,18,023)'}
	P023: INT;
	
	//(18.024) 
	{attribute 'get_bitaccess' := 'ReadUserParameterBit(00,18,024,BITNR)'}
	{attribute 'get_access' := 'ReadUserParameterINT(00,18,024)'}
	{attribute 'set_bitaccess' := 'WriteUserParameterBit(00,18,024,BITNR,P024)'}
	{attribute 'set_access' := 'WriteUserParameterINT(00,18,024,P024)'}
	{attribute 'monitoring_instead' := 'ReadUserParameterINT(00,18,024)'}
	P024: INT;
	
	//(18.025)
	{attribute 'get_bitaccess' := 'ReadUserParameterBit(00,18,025,BITNR)'}
	{attribute 'get_access' := 'ReadUserParameterINT(00,18,025)'}
	{attribute 'set_bitaccess' := 'WriteUserParameterBit(00,18,025,BITNR,P025)'}
	{attribute 'set_access' := 'WriteUserParameterINT(00,18,025,P025)'}
	{attribute 'monitoring_instead' := 'ReadUserParameterINT(00,18,025)'}
	P025: INT;
	
	//(18.026)
	{attribute 'get_bitaccess' := 'ReadUserParameterBit(00,18,026,BITNR)'}
	{attribute 'get_access' := 'ReadUserParameterINT(00,18,026)'}
	{attribute 'set_bitaccess' := 'WriteUserParameterBit(00,18,026,BITNR,P026)'}
	{attribute 'set_access' := 'WriteUserParameterINT(00,18,026,P026)'}
	{attribute 'monitoring_instead' := 'ReadUserParameterINT(00,18,026)'}
	P026: INT;
	
	//(18.027)
	{attribute 'get_bitaccess' := 'ReadUserParameterBit(00,18,027,BITNR)'}
	{attribute 'get_access' := 'ReadUserParameterINT(00,18,027)'}
	{attribute 'set_bitaccess' := 'WriteUserParameterBit(00,18,027,BITNR,P027)'}
	{attribute 'set_access' := 'WriteUserParameterINT(00,18,027,P027)'}
	{attribute 'monitoring_instead' := 'ReadUserParameterINT(00,18,027)'}
	P027: INT;
	
	//(18.028)
	{attribute 'get_bitaccess' := 'ReadUserParameterBit(00,18,028,BITNR)'}
	{attribute 'get_access' := 'ReadUserParameterINT(00,18,028)'}
	{attribute 'set_bitaccess' := 'WriteUserParameterBit(00,18,028,BITNR,P028)'}
	{attribute 'set_access' := 'WriteUserParameterINT(00,18,028,P028)'}
	{attribute 'monitoring_instead' := 'ReadUserParameterINT(00,18,028)'}
	P028: INT;
	
	//(18.029)
	{attribute 'get_bitaccess' := 'ReadUserParameterBit(00,18,029,BITNR)'}
	{attribute 'get_access' := 'ReadUserParameterINT(00,18,029)'}
	{attribute 'set_bitaccess' := 'WriteUserParameterBit(00,18,029,BITNR,P029)'}
	{attribute 'set_access' := 'WriteUserParameterINT(00,18,029,P029)'}
	{attribute 'monitoring_instead' := 'ReadUserParameterINT(00,18,029)'}
	P029: INT;
	
	//(18.030)
	{attribute 'get_bitaccess' := 'ReadUserParameterBit(00,18,030,BITNR)'}
	{attribute 'get_access' := 'ReadUserParameterINT(00,18,030)'}
	{attribute 'set_bitaccess' := 'WriteUserParameterBit(00,18,030,BITNR,P030)'}
	{attribute 'set_access' := 'WriteUserParameterINT(00,18,030,P030)'}
	{attribute 'monitoring_instead' := 'ReadUserParameterINT(00,18,030)'}
	P030: INT;
	
	//(18.031) 
	{attribute 'get_access' := 'ReadUserParameterBOOL(00,18,031)'} 
	{attribute 'set_access' := 'WriteUserParameterBOOL(00,18,031,P031)'}
	{attribute 'monitoring_instead' := 'ReadUserParameterBOOL(00,18,031)'}
	P031: BOOL;
	
	//(18.032) 
	{attribute 'get_access' := 'ReadUserParameterBOOL(00,18,032)'} 
	{attribute 'set_access' := 'WriteUserParameterBOOL(00,18,032,P032)'}
	{attribute 'monitoring_instead' := 'ReadUserParameterBOOL(00,18,032)'}
	P032: BOOL;
	
	//(18.033) 
	{attribute 'get_access' := 'ReadUserParameterBOOL(00,18,033)'} 
	{attribute 'set_access' := 'WriteUserParameterBOOL(00,18,033,P033)'}
	{attribute 'monitoring_instead' := 'ReadUserParameterBOOL(00,18,033)'}
	P033: BOOL;
	
	//(18.034) 
	{attribute 'get_access' := 'ReadUserParameterBOOL(00,18,034)'} 
	{attribute 'set_access' := 'WriteUserParameterBOOL(00,18,034,P034)'}
	{attribute 'monitoring_instead' := 'ReadUserParameterBOOL(00,18,034)'}
	P034: BOOL;
	
	//(18.035) 
	{attribute 'get_access' := 'ReadUserParameterBOOL(00,18,035)'} 
	{attribute 'set_access' := 'WriteUserParameterBOOL(00,18,035,P035)'}
	{attribute 'monitoring_instead' := 'ReadUserParameterBOOL(00,18,035)'}
	P035: BOOL;
	
	//(18.036) 
	{attribute 'get_access' := 'ReadUserParameterBOOL(00,18,036)'} 
	{attribute 'set_access' := 'WriteUserParameterBOOL(00,18,036,P036)'}
	{attribute 'monitoring_instead' := 'ReadUserParameterBOOL(00,18,036)'}
	P036: BOOL;
	
	//(18.037)  
	{attribute 'get_access' := 'ReadUserParameterBOOL(00,18,037)'} 
	{attribute 'set_access' := 'WriteUserParameterBOOL(00,18,037,P037)'}
	{attribute 'monitoring_instead' := 'ReadUserParameterBOOL(00,18,037)'}
	P037: BOOL;
	
	//(18.038)  
	{attribute 'get_access' := 'ReadUserParameterBOOL(00,18,038)'} 
	{attribute 'set_access' := 'WriteUserParameterBOOL(00,18,038,P038)'}
	{attribute 'monitoring_instead' := 'ReadUserParameterBOOL(00,18,038)'}
	P038: BOOL;
	
	//(18.039)
	{attribute 'get_access' := 'ReadUserParameterBOOL(00,18,039)'} 
	{attribute 'set_access' := 'WriteUserParameterBOOL(00,18,039,P039)'}
	{attribute 'monitoring_instead' := 'ReadUserParameterBOOL(00,18,039)'}
	P039: BOOL;
	
	//(18.040)
	{attribute 'get_access' := 'ReadUserParameterBOOL(00,18,040)'} 
	{attribute 'set_access' := 'WriteUserParameterBOOL(00,18,040,P040)'}
	{attribute 'monitoring_instead' := 'ReadUserParameterBOOL(00,18,040)'}
	P040: BOOL;
	
	//(18.041) 
	{attribute 'get_access' := 'ReadUserParameterBOOL(00,18,041)'} 
	{attribute 'set_access' := 'WriteUserParameterBOOL(00,18,041,P041)'}
	{attribute 'monitoring_instead' := 'ReadUserParameterBOOL(00,18,041)'}
	P041: BOOL;
	
	//(18.042) 
	{attribute 'get_access' := 'ReadUserParameterBOOL(00,18,042)'} 
	{attribute 'set_access' := 'WriteUserParameterBOOL(00,18,042,P042)'}
	{attribute 'monitoring_instead' := 'ReadUserParameterBOOL(00,18,042)'}
	P042: BOOL;
	
	//(18.043) 
	{attribute 'get_access' := 'ReadUserParameterBOOL(00,18,043)'} 
	{attribute 'set_access' := 'WriteUserParameterBOOL(00,18,043,P043)'}
	{attribute 'monitoring_instead' := 'ReadUserParameterBOOL(00,18,043)'}
	P043: BOOL;
	
	//(18.044) 
	{attribute 'get_access' := 'ReadUserParameterBOOL(00,18,044)'} 
	{attribute 'set_access' := 'WriteUserParameterBOOL(00,18,044,P044)'}
	{attribute 'monitoring_instead' := 'ReadUserParameterBOOL(00,18,044)'}
	P044: BOOL;
	
	//18.045) 
	{attribute 'get_access' := 'ReadUserParameterBOOL(00,18,045)'} 
	{attribute 'set_access' := 'WriteUserParameterBOOL(00,18,045,P045)'}
	{attribute 'monitoring_instead' := 'ReadUserParameterBOOL(00,18,045)'}
	P045: BOOL;
	
	//(18.046) 
	{attribute 'get_access' := 'ReadUserParameterBOOL(00,18,046)'} 
	{attribute 'set_access' := 'WriteUserParameterBOOL(00,18,046,P046)'}
	{attribute 'monitoring_instead' := 'ReadUserParameterBOOL(00,18,046)'}
	P046: BOOL;
	
	//(18.047) 
	{attribute 'get_access' := 'ReadUserParameterBOOL(00,18,047)'} 
	{attribute 'set_access' := 'WriteUserParameterBOOL(00,18,047,P047)'}
	{attribute 'monitoring_instead' := 'ReadUserParameterBOOL(00,18,047)'}
	P047: BOOL;
	
	//(18.048)  
	{attribute 'get_access' := 'ReadUserParameterBOOL(00,18,048)'} 
	{attribute 'set_access' := 'WriteUserParameterBOOL(00,18,048,P048)'}
	{attribute 'monitoring_instead' := 'ReadUserParameterBOOL(00,18,048)'}
	P048: BOOL;
	
	//(18.049) 
	{attribute 'get_access' := 'ReadUserParameterBOOL(00,18,049)'} 
	{attribute 'set_access' := 'WriteUserParameterBOOL(00,18,049,P049)'}
	{attribute 'monitoring_instead' := 'ReadUserParameterBOOL(00,18,049)'}
	P049: BOOL;
	
	//(18.050)  
	{attribute 'get_access' := 'ReadUserParameterBOOL(00,18,050)'} 
	{attribute 'set_access' := 'WriteUserParameterBOOL(00,18,050,P050)'}
	{attribute 'monitoring_instead' := 'ReadUserParameterBOOL(00,18,050)'}
	P050: BOOL;
	
	//(18.051) 
	{attribute 'get_bitaccess' := 'ReadUserParameterBit(00,18,051,BITNR)'}
	{attribute 'get_access' := 'ReadUserParameterDINT(00,18,051)'}
	{attribute 'set_bitaccess' := 'WriteUserParameterBit(00,18,051,BITNR,Distance_Per_Motor_Turn)'}
	{attribute 'set_access' := 'WriteUserParameterDINT(00,18,051,Distance_Per_Motor_Turn)'}
	{attribute 'monitoring_instead' := 'ReadUserParameterDINT(00,18,051)'}
	Distance_Per_Motor_Turn: DINT := 25;
	
	//(18.052) 
	{attribute 'get_bitaccess' := 'ReadUserParameterBit(00,18,052,BITNR)'}
	{attribute 'get_access' := 'ReadUserParameterDINT(00,18,052)'}
	{attribute 'set_bitaccess' := 'WriteUserParameterBit(00,18,052,BITNR,Distance_Per_Encoder_Turn)'}
	{attribute 'set_access' := 'WriteUserParameterDINT(00,18,052,Distance_Per_Encoder_Turn)'}
	{attribute 'monitoring_instead' := 'ReadUserParameterDINT(00,18,052)'}
	Distance_Per_Encoder_Turn: DINT := 360;
	
	//18.053) 
	{attribute 'get_bitaccess' := 'ReadUserParameterBit(00,18,053,BITNR)'}
	{attribute 'get_access' := 'ReadUserParameterDINT(00,18,053)'}
	{attribute 'set_bitaccess' := 'WriteUserParameterBit(00,18,053,BITNR,Acceleration_Position)'}
	{attribute 'set_access' := 'WriteUserParameterDINT(00,18,053,Acceleration_Position)'}
	{attribute 'monitoring_instead' := 'ReadUserParameterDINT(00,18,053)'}
	Acceleration_Position: DINT := 100;
	

	//(18.054) 
	{attribute 'get_bitaccess' := 'ReadUserParameterBit(00,18,054,BITNR)'}
	{attribute 'get_access' := 'ReadUserParameterDINT(00,18,054)'}
	{attribute 'set_bitaccess' := 'WriteUserParameterBit(00,18,054,BITNR,Decceleration_Position)'}
	{attribute 'set_access' := 'WriteUserParameterDINT(00,18,054,Decceleration_Position)'}
	{attribute 'monitoring_instead' := 'ReadUserParameterDINT(00,18,054)'}
	Decceleration_Position: DINT := 100;
	
END_VAR

// Drive/Application/Variables/AMC Variables/gvAMC_Cam
{attribute 'qualified_only'}
VAR_GLOBAL
	  
	//(35.007) Displays which index in the Cam table the Cam controller is using
	//Update Rate 4ms
	{attribute 'get_access' := 'ReadUserParameterINT(00,35,007)'}
	{attribute 'monitoring_instead' := 'ReadUserParameterINT(00,35,007)'}
	Segment_Index: INT;
  
	//(35.008) Displays the position in the segment that the cam controller is using
	//Update Rate 4ms
	{attribute 'get_access' := 'ReadUserParameterDINT(00,35,008)'}
	{attribute 'monitoring_instead' := 'ReadUserParameterDINT(00,35,008)'}
	Position_In_Segment: DINT;
 
	//(35.010) Displays when the cam controller reaches the end of the cam table
	//Update Rate 4ms
	{attribute 'get_access' := 'ReadUserParameterBOOL(00,35,010)'}
	{attribute 'monitoring_instead' := 'ReadUserParameterBOOL(00,35,010)'}
	Cam_Complete: BOOL;
	 
END_VAR

// Drive/Application/Variables/M701 DRIVE /gvDrive_Menu19
(*
	Menu 19
*)
(*	LEVEL 2 SUPPORT
	Only change the variable name after you know how.
	don't add extra white spaces inside the attribute.
*)
(*
	If you change the name of any of them in this list you also have to change the set_access line of code.
	
	Example:
	change P001 to P001_count
	Then you also need to change the attributes
 
	before
	
	{attribute 'get_bitaccess' := 'ReadUserParameterBit(00,19,001,BITNR)'}
	{attribute 'get_access' := 'ReadUserParameterINT(00,19,001)'}
	{attribute 'set_bitaccess' := 'WriteUserParameterBit(00,19,001,BITNR,P001)'}
	{attribute 'set_access' := 'WriteUserParameterINT(00,19,001,P001)'}
	{attribute 'monitoring_instead' := 'ReadUserParameterINT(00,19,001)'}
	P001: INT;
	
	after change 
	
	{attribute 'get_bitaccess' := 'ReadUserParameterBit(00,19,001,BITNR)'}
	{attribute 'get_access' := 'ReadUserParameterINT(00,19,001)'}
	{attribute 'set_bitaccess' := 'WriteUserParameterBit(00,19,001,BITNR,P001_count)'}
	{attribute 'set_access' := 'WriteUserParameterINT(00,19,001,P001_count)'}
	{attribute 'monitoring_instead' := 'ReadUserParameterINT(00,19,001)'}
	P001_count: INT;
	
*)
{attribute 'qualified_only'}
VAR_GLOBAL
 
	
	//(19.001)
	//save on power down
	{attribute 'get_bitaccess' := 'ReadUserParameterBit(00,19,001,BITNR)'}
	{attribute 'get_access' := 'ReadUserParameterINT(00,19,001)'}
	{attribute 'set_bitaccess' := 'WriteUserParameterBit(00,19,001,BITNR,P001)'}
	{attribute 'set_access' := 'WriteUserParameterINT(00,19,001,P001)'}
	{attribute 'monitoring_instead' := 'ReadUserParameterINT(00,19,001)'}
	P001: INT;
	
	//(19.002) 
	{attribute 'get_bitaccess' := 'ReadUserParameterBit(00,19,002,BITNR)'}
	{attribute 'get_access' := 'ReadUserParameterINT(00,19,002)'}
	{attribute 'set_bitaccess' := 'WriteUserParameterBit(00,19,002,BITNR,P002)'}
	{attribute 'set_access' := 'WriteUserParameterINT(00,19,002,P002)'}
	{attribute 'monitoring_instead' := 'ReadUserParameterINT(00,19,002)'}
	P002: INT;
	
	// (19.003) 
	{attribute 'get_bitaccess' := 'ReadUserParameterBit(00,19,003,BITNR)'}
	{attribute 'get_access' := 'ReadUserParameterINT(00,19,003)'}
	{attribute 'set_bitaccess' := 'WriteUserParameterBit(00,19,003,BITNR,P003)'}
	{attribute 'set_access' := 'WriteUserParameterINT(00,19,003,P003)'}
	{attribute 'monitoring_instead' := 'ReadUserParameterINT(00,19,003)'}
	P003: INT;
	
	//(19.004) 
	{attribute 'get_bitaccess' := 'ReadUserParameterBit(00,19,004,BITNR)'}
	{attribute 'get_access' := 'ReadUserParameterINT(00,19,004)'}
	{attribute 'set_bitaccess' := 'WriteUserParameterBit(00,19,004,BITNR,P004)'}
	{attribute 'set_access' := 'WriteUserParameterINT(00,19,004,P004)'}
	{attribute 'monitoring_instead' := 'ReadUserParameterINT(00,19,004)'}
	P004: INT;
	
	//(19.005) 
	{attribute 'get_bitaccess' := 'ReadUserParameterBit(00,19,005,BITNR)'}
	{attribute 'get_access' := 'ReadUserParameterINT(00,19,005)'}
	{attribute 'set_bitaccess' := 'WriteUserParameterBit(00,19,005,BITNR,P005)'}
	{attribute 'set_access' := 'WriteUserParameterINT(00,19,005,P005)'}
	{attribute 'monitoring_instead' := 'ReadUserParameterINT(00,19,005)'}
	P005: INT;
	
	//(19.006) 
	{attribute 'get_bitaccess' := 'ReadUserParameterBit(00,19,006,BITNR)'}
	{attribute 'get_access' := 'ReadUserParameterINT(00,19,006)'}
	{attribute 'set_bitaccess' := 'WriteUserParameterBit(00,19,006,BITNR,P006)'}
	{attribute 'set_access' := 'WriteUserParameterINT(00,19,006,P006)'}
	{attribute 'monitoring_instead' := 'ReadUserParameterINT(00,19,006)'}
	P006: INT;
	
	//(19.007) 
	{attribute 'get_bitaccess' := 'ReadUserParameterBit(00,19,007,BITNR)'}
	{attribute 'get_access' := 'ReadUserParameterINT(00,19,007)'}
	{attribute 'set_bitaccess' := 'WriteUserParameterBit(00,19,007,BITNR,P007)'}
	{attribute 'set_access' := 'WriteUserParameterINT(00,19,007,P007)'}
	{attribute 'monitoring_instead' := 'ReadUserParameterINT(00,19,007)'}
	P007: INT;
	
	//(19.008)
	{attribute 'get_bitaccess' := 'ReadUserParameterBit(00,19,008,BITNR)'}
	{attribute 'get_access' := 'ReadUserParameterINT(00,19,008)'}
	{attribute 'set_bitaccess' := 'WriteUserParameterBit(00,19,008,BITNR,P008)'}
	{attribute 'set_access' := 'WriteUserParameterINT(00,19,008,P008)'}
	{attribute 'monitoring_instead' := 'ReadUserParameterINT(00,19,008)'}
	P008: INT;
	
	//(19.009)
	{attribute 'get_bitaccess' := 'ReadUserParameterBit(00,19,009,BITNR)'}
	{attribute 'get_access' := 'ReadUserParameterINT(00,19,009)'}
	{attribute 'set_bitaccess' := 'WriteUserParameterBit(00,19,009,BITNR,P009)'}
	{attribute 'set_access' := 'WriteUserParameterINT(00,19,009,P009)'}
	{attribute 'monitoring_instead' := 'ReadUserParameterINT(00,19,009)'}
	P009: INT;
	
	//(19.010) 
	{attribute 'get_bitaccess' := 'ReadUserParameterBit(00,19,010,BITNR)'}
	{attribute 'get_access' := 'ReadUserParameterINT(00,19,010)'}
	{attribute 'set_bitaccess' := 'WriteUserParameterBit(00,19,010,BITNR,P010)'}
	{attribute 'set_access' := 'WriteUserParameterINT(00,19,010,P010)'}
	{attribute 'monitoring_instead' := 'ReadUserParameterINT(00,19,010)'}
	P010: INT;
	
	//(19.011) 
	{attribute 'get_bitaccess' := 'ReadUserParameterBit(00,19,011,BITNR)'}
	{attribute 'get_access' := 'ReadUserParameterINT(00,19,011)'}
	{attribute 'set_bitaccess' := 'WriteUserParameterBit(00,19,011,BITNR,P011)'}
	{attribute 'set_access' := 'WriteUserParameterINT(00,19,011,P011)'}
	{attribute 'monitoring_instead' := 'ReadUserParameterINT(00,19,011)'}
	P011: INT;
	
	//(19.012) 
	{attribute 'get_bitaccess' := 'ReadUserParameterBit(00,19,012,BITNR)'}
	{attribute 'get_access' := 'ReadUserParameterINT(00,19,012)'}
	{attribute 'set_bitaccess' := 'WriteUserParameterBit(00,19,012,BITNR,P012)'}
	{attribute 'set_access' := 'WriteUserParameterINT(00,19,012,P012)'}
	{attribute 'monitoring_instead' := 'ReadUserParameterINT(00,19,012)'}
	P012: INT;
	
	//(19.013) 
	{attribute 'get_bitaccess' := 'ReadUserParameterBit(00,19,013,BITNR)'}
	{attribute 'get_access' := 'ReadUserParameterINT(00,19,013)'}
	{attribute 'set_bitaccess' := 'WriteUserParameterBit(00,19,013,BITNR,P013)'}
	{attribute 'set_access' := 'WriteUserParameterINT(00,19,013,P013)'}
	{attribute 'monitoring_instead' := 'ReadUserParameterINT(00,19,013)'}
	P013: INT;
	
	//(19.014) 
	{attribute 'get_bitaccess' := 'ReadUserParameterBit(00,19,014,BITNR)'}
	{attribute 'get_access' := 'ReadUserParameterINT(00,19,014)'}
	{attribute 'set_bitaccess' := 'WriteUserParameterBit(00,19,014,BITNR,P014)'}
	{attribute 'set_access' := 'WriteUserParameterINT(00,19,014,P014)'}
	{attribute 'monitoring_instead' := 'ReadUserParameterINT(00,19,014)'}
	P014: INT;
	
	//(19.015)
	{attribute 'get_bitaccess' := 'ReadUserParameterBit(00,19,015,BITNR)'}
	{attribute 'get_access' := 'ReadUserParameterINT(00,19,015)'}
	{attribute 'set_bitaccess' := 'WriteUserParameterBit(00,19,015,BITNR,P015)'}
	{attribute 'set_access' := 'WriteUserParameterINT(00,19,015,P015)'}
	{attribute 'monitoring_instead' := 'ReadUserParameterINT(00,19,015)'}
	P015: INT;
	
	//(19.016)
	{attribute 'get_bitaccess' := 'ReadUserParameterBit(00,19,016,BITNR)'}
	{attribute 'get_access' := 'ReadUserParameterINT(00,19,016)'}
	{attribute 'set_bitaccess' := 'WriteUserParameterBit(00,19,016,BITNR,P016)'}
	{attribute 'set_access' := 'WriteUserParameterINT(00,19,016,P016)'}
	{attribute 'monitoring_instead' := 'ReadUserParameterINT(00,19,016)'}
	P016: INT;
	
	//(19.017)
	{attribute 'get_bitaccess' := 'ReadUserParameterBit(00,19,017,BITNR)'}
	{attribute 'get_access' := 'ReadUserParameterINT(00,19,017)'}
	{attribute 'set_bitaccess' := 'WriteUserParameterBit(00,19,017,BITNR,P017)'}
	{attribute 'set_access' := 'WriteUserParameterINT(00,19,017,P017)'}
	{attribute 'monitoring_instead' := 'ReadUserParameterINT(00,19,017)'}
	P017: INT;
	
	//(19.018)
	{attribute 'get_bitaccess' := 'ReadUserParameterBit(00,19,018,BITNR)'}
	{attribute 'get_access' := 'ReadUserParameterINT(00,19,018)'}
	{attribute 'set_bitaccess' := 'WriteUserParameterBit(00,19,018,BITNR,P018)'}
	{attribute 'set_access' := 'WriteUserParameterINT(00,19,019,P018)'}
	{attribute 'monitoring_instead' := 'ReadUserParameterINT(00,19,018)'}
	P018: INT;
	
	//(19.019) 
	{attribute 'get_bitaccess' := 'ReadUserParameterBit(00,19,019,BITNR)'}
	{attribute 'get_access' := 'ReadUserParameterINT(00,19,019)'}
	{attribute 'set_bitaccess' := 'WriteUserParameterBit(00,19,019,BITNR,P019)'}
	{attribute 'set_access' := 'WriteUserParameterINT(00,19,019,P019)'}
	{attribute 'monitoring_instead' := 'ReadUserParameterINT(00,19,019)'}
	P019: INT;
	
	//(19.020)
	{attribute 'get_bitaccess' := 'ReadUserParameterBit(00,19,020,BITNR)'}
	{attribute 'get_access' := 'ReadUserParameterINT(00,19,020)'}
	{attribute 'set_bitaccess' := 'WriteUserParameterBit(00,19,020,BITNR,P020)'}
	{attribute 'set_access' := 'WriteUserParameterINT(00,19,020,P020)'}
	{attribute 'monitoring_instead' := 'ReadUserParameterINT(00,19,020)'}
	P020: INT;
	
	//(19.021)
	{attribute 'get_bitaccess' := 'ReadUserParameterBit(00,19,021,BITNR)'}
	{attribute 'get_access' := 'ReadUserParameterINT(00,19,021)'}
	{attribute 'set_bitaccess' := 'WriteUserParameterBit(00,19,021,BITNR,P021)'}
	{attribute 'set_access' := 'WriteUserParameterINT(00,19,021,P021)'}
	{attribute 'monitoring_instead' := 'ReadUserParameterINT(00,19,021)'}
	P021: INT;
	
	//(19.022) 
	{attribute 'get_bitaccess' := 'ReadUserParameterBit(00,19,022,BITNR)'}
	{attribute 'get_access' := 'ReadUserParameterINT(00,19,022)'}
	{attribute 'set_bitaccess' := 'WriteUserParameterBit(00,19,022,BITNR,P022)'}
	{attribute 'set_access' := 'WriteUserParameterINT(00,19,022,P022)'}
	{attribute 'monitoring_instead' := 'ReadUserParameterINT(00,19,022)'}
	P022: INT;
	
	//(19.023) 
	{attribute 'get_bitaccess' := 'ReadUserParameterBit(00,19,023,BITNR)'}
	{attribute 'get_access' := 'ReadUserParameterINT(00,19,023)'}
	{attribute 'set_bitaccess' := 'WriteUserParameterBit(00,19,023,BITNR,P023)'}
	{attribute 'set_access' := 'WriteUserParameterINT(00,19,023,P023)'}
	{attribute 'monitoring_instead' := 'ReadUserParameterINT(00,19,023)'}
	P023: INT;
	
	//(19.024) 
	{attribute 'get_bitaccess' := 'ReadUserParameterBit(00,19,024,BITNR)'}
	{attribute 'get_access' := 'ReadUserParameterINT(00,19,024)'}
	{attribute 'set_bitaccess' := 'WriteUserParameterBit(00,19,024,BITNR,P024)'}
	{attribute 'set_access' := 'WriteUserParameterINT(00,19,024,P024)'}
	{attribute 'monitoring_instead' := 'ReadUserParameterINT(00,19,024)'}
	P024: INT;
	
	//(19.025)
	{attribute 'get_bitaccess' := 'ReadUserParameterBit(00,19,025,BITNR)'}
	{attribute 'get_access' := 'ReadUserParameterINT(00,19,025)'}
	{attribute 'set_bitaccess' := 'WriteUserParameterBit(00,19,025,BITNR,P025)'}
	{attribute 'set_access' := 'WriteUserParameterINT(00,19,025,P025)'}
	{attribute 'monitoring_instead' := 'ReadUserParameterINT(00,19,025)'}
	P025: INT;
	
	//(19.026)
	{attribute 'get_bitaccess' := 'ReadUserParameterBit(00,19,026,BITNR)'}
	{attribute 'get_access' := 'ReadUserParameterINT(00,19,026)'}
	{attribute 'set_bitaccess' := 'WriteUserParameterBit(00,19,026,BITNR,P026)'}
	{attribute 'set_access' := 'WriteUserParameterINT(00,19,026,P026)'}
	{attribute 'monitoring_instead' := 'ReadUserParameterINT(00,19,026)'}
	P026: INT;
	
	//(19.027)
	{attribute 'get_bitaccess' := 'ReadUserParameterBit(00,19,027,BITNR)'}
	{attribute 'get_access' := 'ReadUserParameterINT(00,19,027)'}
	{attribute 'set_bitaccess' := 'WriteUserParameterBit(00,19,027,BITNR,P027)'}
	{attribute 'set_access' := 'WriteUserParameterINT(00,19,027,P027)'}
	{attribute 'monitoring_instead' := 'ReadUserParameterINT(00,19,027)'}
	P027: INT;
	
	//(19.028)
	{attribute 'get_bitaccess' := 'ReadUserParameterBit(00,19,028,BITNR)'}
	{attribute 'get_access' := 'ReadUserParameterINT(00,19,028)'}
	{attribute 'set_bitaccess' := 'WriteUserParameterBit(00,19,028,BITNR,P028)'}
	{attribute 'set_access' := 'WriteUserParameterINT(00,19,028,P028)'}
	{attribute 'monitoring_instead' := 'ReadUserParameterINT(00,19,028)'}
	P028: INT;
	
	//(19.029)
	{attribute 'get_bitaccess' := 'ReadUserParameterBit(00,19,029,BITNR)'}
	{attribute 'get_access' := 'ReadUserParameterINT(00,19,029)'}
	{attribute 'set_bitaccess' := 'WriteUserParameterBit(00,19,029,BITNR,P029)'}
	{attribute 'set_access' := 'WriteUserParameterINT(00,19,029,P029)'}
	{attribute 'monitoring_instead' := 'ReadUserParameterINT(00,19,029)'}
	P029: INT;
	
	//(19.030)
	{attribute 'get_bitaccess' := 'ReadUserParameterBit(00,19,030,BITNR)'}
	{attribute 'get_access' := 'ReadUserParameterINT(00,19,030)'}
	{attribute 'set_bitaccess' := 'WriteUserParameterBit(00,19,030,BITNR,P030)'}
	{attribute 'set_access' := 'WriteUserParameterINT(00,19,030,P030)'}
	{attribute 'monitoring_instead' := 'ReadUserParameterINT(00,19,030)'}
	P030: INT;
	
	//(19.031) 
	{attribute 'get_access' := 'ReadUserParameterBOOL(00,19,031)'} 
	{attribute 'set_access' := 'WriteUserParameterBOOL(00,19,031,P031)'}
	{attribute 'monitoring_instead' := 'ReadUserParameterBOOL(00,19,031)'}
	P031: BOOL;
	
	//(19.032) 
	{attribute 'get_access' := 'ReadUserParameterBOOL(00,19,032)'} 
	{attribute 'set_access' := 'WriteUserParameterBOOL(00,19,032,P032)'}
	{attribute 'monitoring_instead' := 'ReadUserParameterBOOL(00,19,032)'}
	P032: BOOL;
	
	//(19.033) 
	{attribute 'get_access' := 'ReadUserParameterBOOL(00,19,033)'} 
	{attribute 'set_access' := 'WriteUserParameterBOOL(00,19,033,P033)'}
	{attribute 'monitoring_instead' := 'ReadUserParameterBOOL(00,19,033)'}
	P033: BOOL;
	
	//(19.034) 
	{attribute 'get_access' := 'ReadUserParameterBOOL(00,19,034)'} 
	{attribute 'set_access' := 'WriteUserParameterBOOL(00,19,034,P034)'}
	{attribute 'monitoring_instead' := 'ReadUserParameterBOOL(00,19,034)'}
	P034: BOOL;
	
	//(19.035) 
	{attribute 'get_access' := 'ReadUserParameterBOOL(00,19,035)'} 
	{attribute 'set_access' := 'WriteUserParameterBOOL(00,19,035,P035)'}
	{attribute 'monitoring_instead' := 'ReadUserParameterBOOL(00,19,035)'}
	P035: BOOL;
	
	//(19.036) 
	{attribute 'get_access' := 'ReadUserParameterBOOL(00,19,036)'} 
	{attribute 'set_access' := 'WriteUserParameterBOOL(00,19,036,P036)'}
	{attribute 'monitoring_instead' := 'ReadUserParameterBOOL(00,19,036)'}
	P036: BOOL;
	
	//(19.037)  
	{attribute 'get_access' := 'ReadUserParameterBOOL(00,19,037)'} 
	{attribute 'set_access' := 'WriteUserParameterBOOL(00,19,037,P037)'}
	{attribute 'monitoring_instead' := 'ReadUserParameterBOOL(00,19,037)'}
	P037: BOOL;
	
	//(19.038)  
	{attribute 'get_access' := 'ReadUserParameterBOOL(00,19,038)'} 
	{attribute 'set_access' := 'WriteUserParameterBOOL(00,19,038,P038)'}
	{attribute 'monitoring_instead' := 'ReadUserParameterBOOL(00,19,038)'}
	P038: BOOL;
	
	//(19.039)
	{attribute 'get_access' := 'ReadUserParameterBOOL(00,19,039)'} 
	{attribute 'set_access' := 'WriteUserParameterBOOL(00,19,039,P039)'}
	{attribute 'monitoring_instead' := 'ReadUserParameterBOOL(00,19,039)'}
	P039: BOOL;
	
	//(19.040)
	{attribute 'get_access' := 'ReadUserParameterBOOL(00,19,040)'} 
	{attribute 'set_access' := 'WriteUserParameterBOOL(00,19,040,P040)'}
	{attribute 'monitoring_instead' := 'ReadUserParameterBOOL(00,19,040)'}
	P040: BOOL;
	
	//(19.041) 
	{attribute 'get_access' := 'ReadUserParameterBOOL(00,19,041)'} 
	{attribute 'set_access' := 'WriteUserParameterBOOL(00,19,041,P041)'}
	{attribute 'monitoring_instead' := 'ReadUserParameterBOOL(00,19,041)'}
	P041: BOOL;
	
	//(19.042) 
	{attribute 'get_access' := 'ReadUserParameterBOOL(00,19,042)'} 
	{attribute 'set_access' := 'WriteUserParameterBOOL(00,19,042,P042)'}
	{attribute 'monitoring_instead' := 'ReadUserParameterBOOL(00,19,042)'}
	P042: BOOL;
	
	//(19.043) 
	{attribute 'get_access' := 'ReadUserParameterBOOL(00,19,043)'} 
	{attribute 'set_access' := 'WriteUserParameterBOOL(00,19,043,P043)'}
	{attribute 'monitoring_instead' := 'ReadUserParameterBOOL(00,19,043)'}
	P043: BOOL;
	
	//(19.044) 
	{attribute 'get_access' := 'ReadUserParameterBOOL(00,19,044)'} 
	{attribute 'set_access' := 'WriteUserParameterBOOL(00,19,044,P044)'}
	{attribute 'monitoring_instead' := 'ReadUserParameterBOOL(00,19,044)'}
	P044: BOOL;
	
	//19.045) 
	{attribute 'get_access' := 'ReadUserParameterBOOL(00,19,045)'} 
	{attribute 'set_access' := 'WriteUserParameterBOOL(00,19,045,P045)'}
	{attribute 'monitoring_instead' := 'ReadUserParameterBOOL(00,19,045)'}
	P045: BOOL;
	
	//(19.046) 
	{attribute 'get_access' := 'ReadUserParameterBOOL(00,19,046)'} 
	{attribute 'set_access' := 'WriteUserParameterBOOL(00,19,046,P046)'}
	{attribute 'monitoring_instead' := 'ReadUserParameterBOOL(00,19,046)'}
	P046: BOOL;
	
	//(19.047) 
	{attribute 'get_access' := 'ReadUserParameterBOOL(00,19,047)'} 
	{attribute 'set_access' := 'WriteUserParameterBOOL(00,19,047,P047)'}
	{attribute 'monitoring_instead' := 'ReadUserParameterBOOL(00,19,047)'}
	P047: BOOL;
	
	//(19.048)  
	{attribute 'get_access' := 'ReadUserParameterBOOL(00,19,048)'} 
	{attribute 'set_access' := 'WriteUserParameterBOOL(00,19,048,P048)'}
	{attribute 'monitoring_instead' := 'ReadUserParameterBOOL(00,19,048)'}
	P048: BOOL;
	
	//(19.049) 
	{attribute 'get_access' := 'ReadUserParameterBOOL(00,19,049)'} 
	{attribute 'set_access' := 'WriteUserParameterBOOL(00,19,049,P049)'}
	{attribute 'monitoring_instead' := 'ReadUserParameterBOOL(00,19,049)'}
	P049: BOOL;
	
	//(19.050)  
	{attribute 'get_access' := 'ReadUserParameterBOOL(00,19,050)'} 
	{attribute 'set_access' := 'WriteUserParameterBOOL(00,19,050,P050)'}
	{attribute 'monitoring_instead' := 'ReadUserParameterBOOL(00,19,050)'}
	P050: BOOL;
	
	//(19.051) 
	{attribute 'get_bitaccess' := 'ReadUserParameterBit(00,19,051,BITNR)'}
	{attribute 'get_access' := 'ReadUserParameterDINT(00,19,051)'}
	{attribute 'set_bitaccess' := 'WriteUserParameterBit(00,19,051,BITNR,Jog_Acceleration)'}
	{attribute 'set_access' := 'WriteUserParameterDINT(00,19,051,Jog_Acceleration)'}
	{attribute 'monitoring_instead' := 'ReadUserParameterDINT(00,19,051)'}
	Jog_Acceleration: DINT := 100;
	
	//(19.052) 
	{attribute 'get_bitaccess' := 'ReadUserParameterBit(00,19,052,BITNR)'}
	{attribute 'get_access' := 'ReadUserParameterDINT(00,19,052)'}
	{attribute 'set_bitaccess' := 'WriteUserParameterBit(00,19,052,BITNR,Jog_Decceleration)'}
	{attribute 'set_access' := 'WriteUserParameterDINT(00,19,052,Jog_Decceleration)'}
	{attribute 'monitoring_instead' := 'ReadUserParameterDINT(00,19,052)'}
	Jog_Decceleration: DINT := 100;
	
	//19.053) 
	{attribute 'get_bitaccess' := 'ReadUserParameterBit(00,19,053,BITNR)'}
	{attribute 'get_access' := 'ReadUserParameterDINT(00,19,053)'}
	{attribute 'set_bitaccess' := 'WriteUserParameterBit(00,19,053,BITNR,Jog_Speed)'}
	{attribute 'set_access' := 'WriteUserParameterDINT(00,19,053,Jog_Speed)'}
	{attribute 'monitoring_instead' := 'ReadUserParameterDINT(00,19,053)'}
	Jog_Speed: DINT := 50;
	

	//(19.054) 
	{attribute 'get_bitaccess' := 'ReadUserParameterBit(00,19,054,BITNR)'}
	{attribute 'get_access' := 'ReadUserParameterDINT(00,19,054)'}
	{attribute 'set_bitaccess' := 'WriteUserParameterBit(00,19,054,BITNR,P054)'}
	{attribute 'set_access' := 'WriteUserParameterDINT(00,19,054,P054)'}
	{attribute 'monitoring_instead' := 'ReadUserParameterDINT(00,19,054)'}
	P054: DINT;
	
END_VAR

// Drive/Application/Variables/M701 DRIVE /gvDrive_Menu20
(*
	Menu 19
*)
(*	LEVEL 2 SUPPORT
	Only change the variable name after you know how.
	don't add extra white spaces inside the attribute.
*)
(*
	If you change the name of any of them in this list you also have to change the set_access line of code.
	
	Example:
	change P001 to P001_count
	Then you also need to change the attributes
 
	before
	
	{attribute 'get_bitaccess' := 'ReadUserParameterBit(00,20,001,BITNR)'}
	{attribute 'get_access' := 'ReadUserParameterINT(00,20,001)'}
	{attribute 'set_bitaccess' := 'WriteUserParameterBit(00,20,001,BITNR,P001)'}
	{attribute 'set_access' := 'WriteUserParameterINT(00,20,001,P001)'}
	{attribute 'monitoring_instead' := 'ReadUserParameterINT(00,20,001)'}
	P001: INT;
	
	after change 
	
	{attribute 'get_bitaccess' := 'ReadUserParameterBit(00,20,001,BITNR)'}
	{attribute 'get_access' := 'ReadUserParameterINT(00,20,001)'}
	{attribute 'set_bitaccess' := 'WriteUserParameterBit(00,20,001,BITNR,P001_count)'}
	{attribute 'set_access' := 'WriteUserParameterINT(00,20,001,P001_count)'}
	{attribute 'monitoring_instead' := 'ReadUserParameterINT(00,20,001)'}
	P001_count: INT;
	
*)
{attribute 'qualified_only'}
VAR_GLOBAL
 
	 //(20.001)
	{attribute 'get_bitaccess' := 'ReadUserParameterBit(00,20,001,BITNR)'}
	{attribute 'get_access' := 'ReadUserParameterINT(00,20,001)'}
	{attribute 'set_bitaccess' := 'WriteUserParameterBit(00,20,001,BITNR,P001)'}
	{attribute 'set_access' := 'WriteUserParameterINT(00,20,001,P001)'}
	{attribute 'monitoring_instead' := 'ReadUserParameterINT(00,20,001)'}
	P001: INT;
	
	//(20.002) 
	{attribute 'get_bitaccess' := 'ReadUserParameterBit(00,20,002,BITNR)'}
	{attribute 'get_access' := 'ReadUserParameterINT(00,20,002)'}
	{attribute 'set_bitaccess' := 'WriteUserParameterBit(00,20,002,BITNR,P002)'}
	{attribute 'set_access' := 'WriteUserParameterINT(00,20,002,P002)'}
	{attribute 'monitoring_instead' := 'ReadUserParameterINT(00,20,002)'}
	P002: INT;
	
	// (20.003) 
	{attribute 'get_bitaccess' := 'ReadUserParameterBit(00,20,003,BITNR)'}
	{attribute 'get_access' := 'ReadUserParameterINT(00,20,003)'}
	{attribute 'set_bitaccess' := 'WriteUserParameterBit(00,20,003,BITNR,P003)'}
	{attribute 'set_access' := 'WriteUserParameterINT(00,20,003,P003)'}
	{attribute 'monitoring_instead' := 'ReadUserParameterINT(00,20,003)'}
	P003: INT;
	
	//(20.004) 
	{attribute 'get_bitaccess' := 'ReadUserParameterBit(00,20,004,BITNR)'}
	{attribute 'get_access' := 'ReadUserParameterINT(00,20,004)'}
	{attribute 'set_bitaccess' := 'WriteUserParameterBit(00,20,004,BITNR,P004)'}
	{attribute 'set_access' := 'WriteUserParameterINT(00,20,004,P004)'}
	{attribute 'monitoring_instead' := 'ReadUserParameterINT(00,20,004)'}
	P004: INT;
	
	//(20.005) 
	{attribute 'get_bitaccess' := 'ReadUserParameterBit(00,20,005,BITNR)'}
	{attribute 'get_access' := 'ReadUserParameterINT(00,20,005)'}
	{attribute 'set_bitaccess' := 'WriteUserParameterBit(00,20,005,BITNR,P005)'}
	{attribute 'set_access' := 'WriteUserParameterINT(00,20,005,P005)'}
	{attribute 'monitoring_instead' := 'ReadUserParameterINT(00,20,005)'}
	P005: INT;
	
	//(20.006) 
	{attribute 'get_bitaccess' := 'ReadUserParameterBit(00,20,006,BITNR)'}
	{attribute 'get_access' := 'ReadUserParameterINT(00,20,006)'}
	{attribute 'set_bitaccess' := 'WriteUserParameterBit(00,20,006,BITNR,P006)'}
	{attribute 'set_access' := 'WriteUserParameterINT(00,20,006,P006)'}
	{attribute 'monitoring_instead' := 'ReadUserParameterINT(00,20,006)'}
	P006: INT;
	
	//(20.007) 
	{attribute 'get_bitaccess' := 'ReadUserParameterBit(00,20,007,BITNR)'}
	{attribute 'get_access' := 'ReadUserParameterINT(00,20,007)'}
	{attribute 'set_bitaccess' := 'WriteUserParameterBit(00,20,007,BITNR,P007)'}
	{attribute 'set_access' := 'WriteUserParameterINT(00,20,007,P007)'}
	{attribute 'monitoring_instead' := 'ReadUserParameterINT(00,20,007)'}
	P007: INT;
	
	//(20.008)
	{attribute 'get_bitaccess' := 'ReadUserParameterBit(00,20,008,BITNR)'}
	{attribute 'get_access' := 'ReadUserParameterINT(00,20,008)'}
	{attribute 'set_bitaccess' := 'WriteUserParameterBit(00,20,008,BITNR,P008)'}
	{attribute 'set_access' := 'WriteUserParameterINT(00,20,008,P008)'}
	{attribute 'monitoring_instead' := 'ReadUserParameterINT(00,20,008)'}
	P008: INT;
	
	//(20.009)
	{attribute 'get_bitaccess' := 'ReadUserParameterBit(00,20,009,BITNR)'}
	{attribute 'get_access' := 'ReadUserParameterINT(00,20,009)'}
	{attribute 'set_bitaccess' := 'WriteUserParameterBit(00,20,009,BITNR,P009)'}
	{attribute 'set_access' := 'WriteUserParameterINT(00,20,009,P009)'}
	{attribute 'monitoring_instead' := 'ReadUserParameterINT(00,20,009)'}
	P009: INT;
	
	//(20.010) 
	{attribute 'get_bitaccess' := 'ReadUserParameterBit(00,20,010,BITNR)'}
	{attribute 'get_access' := 'ReadUserParameterINT(00,20,010)'}
	{attribute 'set_bitaccess' := 'WriteUserParameterBit(00,20,010,BITNR,P010)'}
	{attribute 'set_access' := 'WriteUserParameterINT(00,20,010,P010)'}
	{attribute 'monitoring_instead' := 'ReadUserParameterINT(00,20,010)'}
	P010: INT;
	
	//(20.011) 
	{attribute 'get_bitaccess' := 'ReadUserParameterBit(00,20,011,BITNR)'}
	{attribute 'get_access' := 'ReadUserParameterINT(00,20,011)'}
	{attribute 'set_bitaccess' := 'WriteUserParameterBit(00,20,011,BITNR,P011)'}
	{attribute 'set_access' := 'WriteUserParameterINT(00,20,011,P011)'}
	{attribute 'monitoring_instead' := 'ReadUserParameterINT(00,20,011)'}
	P011: INT;
	
	//(20.012) 
	{attribute 'get_bitaccess' := 'ReadUserParameterBit(00,20,012,BITNR)'}
	{attribute 'get_access' := 'ReadUserParameterINT(00,20,012)'}
	{attribute 'set_bitaccess' := 'WriteUserParameterBit(00,20,012,BITNR,P012)'}
	{attribute 'set_access' := 'WriteUserParameterINT(00,20,012,P012)'}
	{attribute 'monitoring_instead' := 'ReadUserParameterINT(00,20,012)'}
	P012: INT;
	
	//(20.013) 
	{attribute 'get_bitaccess' := 'ReadUserParameterBit(00,20,013,BITNR)'}
	{attribute 'get_access' := 'ReadUserParameterINT(00,20,013)'}
	{attribute 'set_bitaccess' := 'WriteUserParameterBit(00,20,013,BITNR,P013)'}
	{attribute 'set_access' := 'WriteUserParameterINT(00,20,013,P013)'}
	{attribute 'monitoring_instead' := 'ReadUserParameterINT(00,20,013)'}
	P013: INT;
	
	//(20.014) 
	{attribute 'get_bitaccess' := 'ReadUserParameterBit(00,20,014,BITNR)'}
	{attribute 'get_access' := 'ReadUserParameterINT(00,20,014)'}
	{attribute 'set_bitaccess' := 'WriteUserParameterBit(00,20,014,BITNR,P014)'}
	{attribute 'set_access' := 'WriteUserParameterINT(00,20,014,P014)'}
	{attribute 'monitoring_instead' := 'ReadUserParameterINT(00,20,014)'}
	P014: INT;
	
	//(20.015)
	{attribute 'get_bitaccess' := 'ReadUserParameterBit(00,20,015,BITNR)'}
	{attribute 'get_access' := 'ReadUserParameterINT(00,20,015)'}
	{attribute 'set_bitaccess' := 'WriteUserParameterBit(00,20,015,BITNR,P015)'}
	{attribute 'set_access' := 'WriteUserParameterINT(00,20,015,P015)'}
	{attribute 'monitoring_instead' := 'ReadUserParameterINT(00,20,015)'}
	P015: INT;
	
	//(20.016)
	{attribute 'get_bitaccess' := 'ReadUserParameterBit(00,20,016,BITNR)'}
	{attribute 'get_access' := 'ReadUserParameterINT(00,20,016)'}
	{attribute 'set_bitaccess' := 'WriteUserParameterBit(00,20,016,BITNR,P016)'}
	{attribute 'set_access' := 'WriteUserParameterINT(00,20,016,P016)'}
	{attribute 'monitoring_instead' := 'ReadUserParameterINT(00,20,016)'}
	P016: INT;
	
	//(20.017)
	{attribute 'get_bitaccess' := 'ReadUserParameterBit(00,20,017,BITNR)'}
	{attribute 'get_access' := 'ReadUserParameterINT(00,20,017)'}
	{attribute 'set_bitaccess' := 'WriteUserParameterBit(00,20,017,BITNR,P017)'}
	{attribute 'set_access' := 'WriteUserParameterINT(00,20,017,P017)'}
	{attribute 'monitoring_instead' := 'ReadUserParameterINT(00,20,017)'}
	P017: INT;
	
	//(20.018)
	{attribute 'get_bitaccess' := 'ReadUserParameterBit(00,20,018,BITNR)'}
	{attribute 'get_access' := 'ReadUserParameterINT(00,20,018)'}
	{attribute 'set_bitaccess' := 'WriteUserParameterBit(00,20,018,BITNR,P018)'}
	{attribute 'set_access' := 'WriteUserParameterINT(00,20,020,P018)'}
	{attribute 'monitoring_instead' := 'ReadUserParameterINT(00,20,018)'}
	P018: INT;
	
	//(20.019) 
	{attribute 'get_bitaccess' := 'ReadUserParameterBit(00,20,019,BITNR)'}
	{attribute 'get_access' := 'ReadUserParameterINT(00,20,019)'}
	{attribute 'set_bitaccess' := 'WriteUserParameterBit(00,20,019,BITNR,P020)'}
	{attribute 'set_access' := 'WriteUserParameterINT(00,20,019,P020)'}
	{attribute 'monitoring_instead' := 'ReadUserParameterINT(00,20,019)'}
	P019: INT;
	
	//(20.020)
	{attribute 'get_bitaccess' := 'ReadUserParameterBit(00,20,020,BITNR)'}
	{attribute 'get_access' := 'ReadUserParameterINT(00,20,020)'}
	{attribute 'set_bitaccess' := 'WriteUserParameterBit(00,20,020,BITNR,P020)'}
	{attribute 'set_access' := 'WriteUserParameterINT(00,20,020,P020)'}
	{attribute 'monitoring_instead' := 'ReadUserParameterINT(00,20,020)'}
	P020: INT;
	

	
	
	//(20.021) 
	{attribute 'get_bitaccess' := 'ReadUserParameterBit(00,20,021,BITNR)'}
	{attribute 'get_access' := 'ReadUserParameterDINT(00,20,021)'}
	{attribute 'set_bitaccess' := 'WriteUserParameterBit(00,20,021,BITNR,P021)'}
	{attribute 'set_access' := 'WriteUserParameterDINT(00,20,021,P021)'}
	{attribute 'monitoring_instead' := 'ReadUserParameterDINT(00,20,021)'}
	P021: DINT;
	 
	//(20.022) 
	{attribute 'get_bitaccess' := 'ReadUserParameterBit(00,20,022,BITNR)'}
	{attribute 'get_access' := 'ReadUserParameterDINT(00,20,022)'}
	{attribute 'set_bitaccess' := 'WriteUserParameterBit(00,20,022,BITNR,P022)'}
	{attribute 'set_access' := 'WriteUserParameterDINT(00,20,022,P022)'}
	{attribute 'monitoring_instead' := 'ReadUserParameterDINT(00,20,022)'}
	P022: DINT;
  
	//(20.023) 
	{attribute 'get_bitaccess' := 'ReadUserParameterBit(00,20,023,BITNR)'}
	{attribute 'get_access' := 'ReadUserParameterDINT(00,20,023)'}
	{attribute 'set_bitaccess' := 'WriteUserParameterBit(00,20,023,BITNR,P023)'}
	{attribute 'set_access' := 'WriteUserParameterDINT(00,20,023,P023)'}
	{attribute 'monitoring_instead' := 'ReadUserParameterDINT(00,20,023)'}
	P023: DINT;

	//(20.024) 
	{attribute 'get_bitaccess' := 'ReadUserParameterBit(00,20,024,BITNR)'}
	{attribute 'get_access' := 'ReadUserParameterDINT(00,20,024)'}
	{attribute 'set_bitaccess' := 'WriteUserParameterBit(00,20,024,BITNR,P024)'}
	{attribute 'set_access' := 'WriteUserParameterDINT(00,20,024,P024)'}
	{attribute 'monitoring_instead' := 'ReadUserParameterDINT(00,20,024)'}
	P024: DINT; 
 	
	//(20.025) 
	{attribute 'get_bitaccess' := 'ReadUserParameterBit(00,20,025,BITNR)'}
	{attribute 'get_access' := 'ReadUserParameterDINT(00,20,025)'}
	{attribute 'set_bitaccess' := 'WriteUserParameterBit(00,20,025,BITNR,P025)'}
	{attribute 'set_access' := 'WriteUserParameterDINT(00,20,025,P025)'}
	{attribute 'monitoring_instead' := 'ReadUserParameterDINT(00,20,025)'}
	P025: DINT; 
 	
	//(20.026) 
	{attribute 'get_bitaccess' := 'ReadUserParameterBit(00,20,026,BITNR)'}
	{attribute 'get_access' := 'ReadUserParameterDINT(00,20,026)'}
	{attribute 'set_bitaccess' := 'WriteUserParameterBit(00,20,026,BITNR,P026)'}
	{attribute 'set_access' := 'WriteUserParameterDINT(00,20,026,P026)'}
	{attribute 'monitoring_instead' := 'ReadUserParameterDINT(00,20,026)'}
	P026: DINT; 
 
	//(20.027) 
	{attribute 'get_bitaccess' := 'ReadUserParameterBit(00,20,027,BITNR)'}
	{attribute 'get_access' := 'ReadUserParameterDINT(00,20,027)'}
	{attribute 'set_bitaccess' := 'WriteUserParameterBit(00,20,027,BITNR,P027)'}
	{attribute 'set_access' := 'WriteUserParameterDINT(00,20,027,P027)'}
	{attribute 'monitoring_instead' := 'ReadUserParameterDINT(00,20,027)'}
	P027: DINT;  

	//(20.028) 
	{attribute 'get_bitaccess' := 'ReadUserParameterBit(00,20,028,BITNR)'}
	{attribute 'get_access' := 'ReadUserParameterDINT(00,20,028)'}
	{attribute 'set_bitaccess' := 'WriteUserParameterBit(00,20,028,BITNR,P028)'}
	{attribute 'set_access' := 'WriteUserParameterDINT(00,20,028,P028)'}
	{attribute 'monitoring_instead' := 'ReadUserParameterDINT(00,20,028)'}
	P028: DINT;
  
	//(20.029) 
	{attribute 'get_bitaccess' := 'ReadUserParameterBit(00,20,029,BITNR)'}
	{attribute 'get_access' := 'ReadUserParameterDINT(00,20,029)'}
	{attribute 'set_bitaccess' := 'WriteUserParameterBit(00,20,029,BITNR,P029)'}
	{attribute 'set_access' := 'WriteUserParameterDINT(00,20,029,P029)'}
	{attribute 'monitoring_instead' := 'ReadUserParameterDINT(00,20,029)'}
	P029: DINT;  	

	//(20.030) 
	{attribute 'get_bitaccess' := 'ReadUserParameterBit(00,20,030,BITNR)'}
	{attribute 'get_access' := 'ReadUserParameterDINT(00,20,030)'}
	{attribute 'set_bitaccess' := 'WriteUserParameterBit(00,20,030,BITNR,P030)'}
	{attribute 'set_access' := 'WriteUserParameterDINT(00,20,030,P030)'}
	{attribute 'monitoring_instead' := 'ReadUserParameterDINT(00,20,030)'}
	P030: DINT;  	

	//(20.031) 
	{attribute 'get_bitaccess' := 'ReadUserParameterBit(00,20,031,BITNR)'}
	{attribute 'get_access' := 'ReadUserParameterDINT(00,20,031)'}
	{attribute 'set_bitaccess' := 'WriteUserParameterBit(00,20,031,BITNR,P031)'}
	{attribute 'set_access' := 'WriteUserParameterDINT(00,20,031,P031)'}
	{attribute 'monitoring_instead' := 'ReadUserParameterDINT(00,20,031)'}
	P031: DINT; 
 	
	//(20.032) 
	{attribute 'get_bitaccess' := 'ReadUserParameterBit(00,20,032,BITNR)'}
	{attribute 'get_access' := 'ReadUserParameterDINT(00,20,032)'}
	{attribute 'set_bitaccess' := 'WriteUserParameterBit(00,20,032,BITNR,P032)'}
	{attribute 'set_access' := 'WriteUserParameterDINT(00,20,032,P032)'}
	{attribute 'monitoring_instead' := 'ReadUserParameterDINT(00,20,032)'}
	P032: DINT; 
 	
	//(20.033) 
	{attribute 'get_bitaccess' := 'ReadUserParameterBit(00,20,033,BITNR)'}
	{attribute 'get_access' := 'ReadUserParameterDINT(00,20,033)'}
	{attribute 'set_bitaccess' := 'WriteUserParameterBit(00,20,033,BITNR,P033)'}
	{attribute 'set_access' := 'WriteUserParameterDINT(00,20,033,P033)'}
	{attribute 'monitoring_instead' := 'ReadUserParameterDINT(00,20,033)'}
	P033: DINT; 
 	
	//(20.034) 
	{attribute 'get_bitaccess' := 'ReadUserParameterBit(00,20,034,BITNR)'}
	{attribute 'get_access' := 'ReadUserParameterDINT(00,20,034)'}
	{attribute 'set_bitaccess' := 'WriteUserParameterBit(00,20,034,BITNR,P034)'}
	{attribute 'set_access' := 'WriteUserParameterDINT(00,20,034,P034)'}
	{attribute 'monitoring_instead' := 'ReadUserParameterDINT(00,20,034)'}
	P034: DINT; 
 	
	//(20.035) 
	{attribute 'get_bitaccess' := 'ReadUserParameterBit(00,20,035,BITNR)'}
	{attribute 'get_access' := 'ReadUserParameterDINT(00,20,035)'}
	{attribute 'set_bitaccess' := 'WriteUserParameterBit(00,20,035,BITNR,P035)'}
	{attribute 'set_access' := 'WriteUserParameterDINT(00,20,035,P035)'}
	{attribute 'monitoring_instead' := 'ReadUserParameterDINT(00,20,035)'}
	P035: DINT; 
 	
	//(20.036) 
	{attribute 'get_bitaccess' := 'ReadUserParameterBit(00,20,036,BITNR)'}
	{attribute 'get_access' := 'ReadUserParameterDINT(00,20,036)'}
	{attribute 'set_bitaccess' := 'WriteUserParameterBit(00,20,036,BITNR,P036)'}
	{attribute 'set_access' := 'WriteUserParameterDINT(00,20,036,P036)'}
	{attribute 'monitoring_instead' := 'ReadUserParameterDINT(00,20,036)'}
	P036: DINT;  	

	//(20.037) 
	{attribute 'get_bitaccess' := 'ReadUserParameterBit(00,20,037,BITNR)'}
	{attribute 'get_access' := 'ReadUserParameterDINT(00,20,037)'}
	{attribute 'set_bitaccess' := 'WriteUserParameterBit(00,20,037,BITNR,P037)'}
	{attribute 'set_access' := 'WriteUserParameterDINT(00,20,037,P037)'}
	{attribute 'monitoring_instead' := 'ReadUserParameterDINT(00,20,037)'}
	P037: DINT;  	

	//(20.038) 
	{attribute 'get_bitaccess' := 'ReadUserParameterBit(00,20,038,BITNR)'}
	{attribute 'get_access' := 'ReadUserParameterDINT(00,20,038)'}
	{attribute 'set_bitaccess' := 'WriteUserParameterBit(00,20,038,BITNR,P038)'}
	{attribute 'set_access' := 'WriteUserParameterDINT(00,20,038,P038)'}
	{attribute 'monitoring_instead' := 'ReadUserParameterDINT(00,20,038)'}
	P038: DINT;  	

	//(20.039) 
	{attribute 'get_bitaccess' := 'ReadUserParameterBit(00,20,039,BITNR)'}
	{attribute 'get_access' := 'ReadUserParameterDINT(00,20,039)'}
	{attribute 'set_bitaccess' := 'WriteUserParameterBit(00,20,039,BITNR,P039)'}
	{attribute 'set_access' := 'WriteUserParameterDINT(00,20,039,P039)'}
	{attribute 'monitoring_instead' := 'ReadUserParameterDINT(00,20,039)'}
	P039: DINT; 	

	//(20.040) 
	{attribute 'get_bitaccess' := 'ReadUserParameterBit(00,20,040,BITNR)'}
	{attribute 'get_access' := 'ReadUserParameterDINT(00,20,040)'}
	{attribute 'set_bitaccess' := 'WriteUserParameterBit(00,20,040,BITNR,P040)'}
	{attribute 'set_access' := 'WriteUserParameterDINT(00,20,040,P040)'}
	{attribute 'monitoring_instead' := 'ReadUserParameterDINT(00,20,040)'}
	P040: DINT;
 
 
 
 
 
 
 
 
 
 
 
 
 
 
 
	
END_VAR

// Drive/Application/Variables/M701 DRIVE /gvDrive_Digital_Inverts
(*
	If you change the name of the inverts in this list you also have to change the set_access line of code.
	
	Example:
	change IO_01 to IO_01_stop
	Then you also need to change
	attribute 'set_access' := 'WriteUserParameterSINT(00,08,011,IO_01)'
	to
	attribute 'set_access' := 'WriteUserParameterSINT(00,08,011,IO_01_stop)'
	
*)

{attribute 'qualified_only'}
VAR_GLOBAL

	
	// Digital I/O 01 Invert(08.011), range 0-1. Mode(s) All Modes.
    // [Get:Set] Set to invert Digital I/O 01.
    {attribute 'get_access' := 'ReadUserParameterSINT(00,08,011)'}
    {attribute 'set_access' := 'WriteUserParameterSINT(00,08,011,IO_01)'}
    {attribute 'monitoring_instead' := 'ReadUserParameterSINT(00,08,011)'}
    IO_01 : SINT;

    // Digital I/O 02 Invert(08.012), range 0-1. Mode(s) All Modes.
    // [Get:Set] Set to invert Digital I/O 02.
    {attribute 'get_access' := 'ReadUserParameterSINT(00,08,012)'}
    {attribute 'set_access' := 'WriteUserParameterSINT(00,08,012,IO_02)'}
    {attribute 'monitoring_instead' := 'ReadUserParameterSINT(00,08,012)'}
    IO_02 : SINT;

    // Digital I/O 03 Invert(08.013), range 0-1. Mode(s) All Modes.
    // [Get:Set] Set to invert Digital I/O 03.
    {attribute 'get_access' := 'ReadUserParameterSINT(00,08,013)'}
    {attribute 'set_access' := 'WriteUserParameterSINT(00,08,013,IO_03)'}
    {attribute 'monitoring_instead' := 'ReadUserParameterSINT(00,08,013)'}
    IO_03 : SINT;

    // Digital Input 04 Invert(08.014), range 0-1. Mode(s) All Modes.
    // [Get:Set] Set to invert Digital Input 04.
    {attribute 'get_access' := 'ReadUserParameterSINT(00,08,014)'}
    {attribute 'set_access' := 'WriteUserParameterSINT(00,08,014,Input04)'}
    {attribute 'monitoring_instead' := 'ReadUserParameterSINT(00,08,014)'}
    Input04 : SINT;

    // Digital Input 05 Invert(08.015), range 0-1. Mode(s) All Modes.
    // [Get:Set] Set to invert Digital Input 05.
    {attribute 'get_access' := 'ReadUserParameterSINT(00,08,015)'}
    {attribute 'set_access' := 'WriteUserParameterSINT(00,08,015,Input05)'}
    {attribute 'monitoring_instead' := 'ReadUserParameterSINT(00,08,015)'}
    Input05 : SINT;

    // Digital Input 06 Invert(08.016), range 0-1. Mode(s) All Modes.
    // [Get:Set] Set to invert Digital Input 06.
    {attribute 'get_access' := 'ReadUserParameterSINT(00,08,016)'}
    {attribute 'set_access' := 'WriteUserParameterSINT(00,08,016,Input06)'}
    {attribute 'monitoring_instead' := 'ReadUserParameterSINT(00,08,016)'}
    Input06 : SINT;

    // Relay Invert(08.017), range 0-1. Mode(s) All Modes.
    // [Get:Set] Set to invert the Relay Output.
    {attribute 'get_access' := 'ReadUserParameterSINT(00,08,017)'}
    {attribute 'set_access' := 'WriteUserParameterSINT(00,08,017,RelayOutput)'}
    {attribute 'monitoring_instead' := 'ReadUserParameterSINT(00,08,017)'}
    RelayOutput : SINT;

    // 24V Supply Output Invert(08.018), range 0-1. Mode(s) All Modes.
    // [Get:Set] Set to invert 24V Supply Output.
    {attribute 'get_access' := 'ReadUserParameterSINT(00,08,018)'}
    {attribute 'set_access' := 'WriteUserParameterSINT(00,08,018,VoltageSupplyOutput)'}
    {attribute 'monitoring_instead' := 'ReadUserParameterSINT(00,08,018)'}
    VoltageSupplyOutput : SINT;

END_VAR

// Drive/Application/Variables/AMC Variables/gvAMC_Speed
{attribute 'qualified_only'}
VAR_GLOBAL
	
  
	
    //(32.005), AMC Master Speed
	//Displays the  rate of change of the AMC Master Position, in user units
    {attribute 'get_access' := 'ReadUserParameterLREAL(00,32,005)'}
    {attribute 'monitoring_instead' := 'ReadUserParameterLREAL(00,32,005)'}
    MasterSpeed : LREAL;
	
	//(33.005), AMC System Speed
    //Displays the rate of change of the AMC Slave Position, in user units
    {attribute 'get_access' := 'ReadUserParameterLREAL(00,33,005)'}
    {attribute 'monitoring_instead' := 'ReadUserParameterLREAL(00,33,005)'}
    SystemSpeed : LREAL;
	
	
END_VAR

// Drive/Application/Basic AMC Library/01 Setup/AMC_Enable
(* 
Just enables the AMC.
Note the Drive must be in Inhibit or this function will Error and not run.
This can be done using the parameters 02.005, 02.050, 31.001,  31.011,  41.001. 


*)
//Version 0.00.03
//Cannon Melville 
FUNCTION AMC_Enable
VAR_INPUT
	
	//Enable The AMC
	bEnable	: BOOL ;  	
 	
END_VAR

VAR_OUTPUT 
	
END_VAR

(*	 
	Editing the code in this function may result in limited support. 	 
*)

(*Notes
	The code below uses fuctions to read and write to the drive.  The fuction format is shown below.
	WriteUserParameterUINT(Slot ,Menu	,Parameter, value );
	Value := ReadUserParameterDINT(Slot  ,Menu	,Parameter );
*)
 

	//******************************Just get the AMC Running*******************************\\

	//Parameter 02.005  Disable Standard Ramp Output
	WriteUserParameterBool(00,02,005,bEnable);
	
	//11.029  Software Version
	//Timing otions set to 8	
	//In firmware 1.13.00.00 and newer this is controlled by the drive. 
	IF ReadUserParameterDINT(00,11,029) < 1130000 THEN		
		WriteUserParameterUINT(00,02,050,8);									//enable the AMC Controller
		//Timing otions active set to 8	 
		//WriteUserParameterUINT(00,02,051,8); 
	END_IF
		
	 
	//Don't let the MCi210 oor MCi200 take control of the drive.
	//This is not needed 
	//WriteUserParameterBOOL(03,06,002,FALSE); 


	//31.001  AMC Select
	//Lets the AMC take control of the drives hard speed reference
	WriteUserParameterBOOL(00,31,001,bEnable);
	
	//31.011  AMC Synchronise To Onboard User Program Clock Task
	//This can be removed.
	WriteUserParameterBOOL(00,31,011,FALSE); 
	
	//41.001  AMC Enable
	//Turn on the AMC controler
	WriteUserParameterBOOL(00,41,001,bEnable);

END_FUNCTION

// Drive/Application/Basic AMC Library/01 Setup/AMC_MasterUnits
(* 
This Block is used to setup the UserUnits of the drive.  
Assumptions list. 
	1. Parameter 3.057, 3.157 = 16 for the normalization turns, or whatever option modules you are using will also have a value of 16 for its normalization setting.	
	2. The Drive is in single loop mode and not duel loop mode.
	3. The units are always based on 1 turn of the encoder.
	4. The drive was default before running these blocks for the first time.
	5. That the User will setup parameters 3.024, 33.001, 32.001 and 39.001*)

//Version 0.00.01
//Cannon Melville
//. 
FUNCTION AMC_MasterUnits

//Input
VAR_INPUT
	//This setting is the distance the load travels in user units per turn of the motor.
	//Distance_Per_Motor_Turn = Distance of load / number of motor turns
	Distance_Per_Encoder_Turn : DINT; 
	
END_VAR
	
//Output
VAR_OUTPUT 
	// This output is here because Continuous Function Chart (CFC) Needs 1 or more outputs. 
	// This output is not needed as it alway outputs FALSE.
	//bError: BOOL;  
END_VAR 

VAR 
	
END_VAR

(*	 
	Editing the code in this function may result in limited support. 	 
*)

(*Notes
	The code below uses fuctions to read and write to the drive.  The fuction format is shown below.
	WriteUserParameterUINT(Slot ,Menu	,Parameter, value );
	Value := ReadUserParameterDINT(Slot  ,Menu	,Parameter );
*) 
 

//31.004  AMC Master User Units Ratio Numerator
//Setup the Numerator  (Units Per revolution)
//THE DRIVES UNITS
WriteUserParameterDINT(00,31,004,Distance_Per_Encoder_Turn);			//Writes to the unit 
		
//31.005  AMC Master User Units Ratio Denominator
//Setup the Denominator 
//A value of 65536 = 1 turn of the motor, if parameter 3.057, 3.157, or what ever normalization turns source you are using equals a value of 16 
WriteUserParameterDINT(00,31,005,65536);
 

//Wait 4ms so the the Drive can see that the values changed.
Wait_Time(T#4MS);

END_FUNCTION

// Drive/Application/Basic AMC Library/10 Other/Wait_Time
//Simple wait block used to cause a delay in the middle of a program.
//Useful for allowing the drive parameters to update before trying to read other parameter.


//Version 0.00.01
//Cannon Melville
FUNCTION Wait_Time : BOOL
VAR_INPUT
	tDelayTime	: TIME;
END_VAR
VAR
	tEndTime	: TIME; 	
END_VAR

(*	 
	Editing the code in this function may result in limited support. 	 
*)

tEndTime	:= TIME() + tDelayTime;

WHILE TIME() < tEndTime DO
	Wait_Time	:= FALSE;
END_WHILE

Wait_Time	:= TRUE;

END_FUNCTION

// Drive/Application/Basic AMC Library/01 Setup/AMC_UserUnits
(* 
This Block is used to setup the UserUnits of the drive.  
Assumptions list. 
	1. Parameter 3.057, 3.157 = 16 for the normalization turns, or whatever option modules you are using will also have a value of 16 for its normalization setting.	
	2. The Drive is in single loop mode and not duel loop mode.
	3. The units are always based on 1 turn of the motor.
	4. The drive was default before running these blocks for the first time.
	5. That the User will setup parameters 3.024, 33.001, 32.001 and 39.001*)

//Version 0.00.13
//Cannon Melville
//. 
FUNCTION AMC_UserUnits

//Input
VAR_INPUT
	//This setting is the distance the load travels in user units per turn of the motor.
	//Distance_Per_Motor_Turn = Distance of load / number of motor turns
	Distance_Per_Motor_Turn : DINT; 
	
END_VAR
	
//Output
VAR_OUTPUT 
	// This output is here because Continuous Function Chart (CFC) Needs 1 or more outputs. 
	// This output is not needed as it alway outputs FALSE.
	//bError: BOOL;
END_VAR 

VAR 
	
END_VAR

(*	 
	Editing the code in this function may result in limited support. 	 
*)

(*Notes
	The code below uses fuctions to read and write to the drive.  The fuction format is shown below.
	WriteUserParameterUINT(Slot ,Menu	,Parameter, value );
	Value := ReadUserParameterDINT(Slot  ,Menu	,Parameter );
*) 
 

//31.006  AMC Slave User Units Ratio Numerator
//Setup the Numerator  (Units Per revolution)
//THE DRIVES UNITS
WriteUserParameterDINT(00,31,006,Distance_Per_Motor_Turn);			//Writes to the unit 
		
//31.007  AMC Slave User Units Ratio Denominator
//Setup the Denominator 
//A value of 65536 = 1 turn of the motor, if parameter 3.057, 3.157, or what ever normalization turns source you are using equals a value of 16 
WriteUserParameterDINT(00,31,007,65536);

//31.008  AMC Output User Units Ratio Numerator
//A value of 65536 = 1 turn of the motor, if parameter 3.057, 3.157, or what ever normalization turns source you are using equals a value of 16 
//This is used to convert the user units in to RPM
//This parameter is used so the drive can be put in dual loop if needed
WriteUserParameterDINT(00,31,008,65536);							//Writes to the Output Numerator.  This is for the ouput of the AMC to the motor speed loop.  Put the units back into RPM
 
//31.009  AMC Output User Units Ratio Denominator 
//This is used to convert the user units into RPM
//This parameter is used so the drive can be put in dual loop if needed
WriteUserParameterDINT(00,31,009,Distance_Per_Motor_Turn);			//Writes to the Output Denominator.  This is for the ouput of the AMC to the motor speed loop.  Put the units back into RPM

//Wait 4ms so the the Drive can see that the values changed.
Wait_Time(T#4MS);

END_FUNCTION

// Drive/Application/Basic AMC Library/01 Setup/AMC_StopMode
(*
This Block is used to setup how the AMC will stop on a stop command.  There are two basic stop commands: standard stop command, and a following error stop command.
Both stop commands are effected by the mode.

Parameter 34.001 is the stop mode parameter.

Value 	Disc 
0 		Profile Stop if the user commands a stop motion command.
1 		No Profile stop if the user commands a stop motion command.
2 		Profile Stop if the user commands a stop motion command or if the position is outside the following error window.
3 		No Profile Stop if the user commands a stop motion command or if the position is outside the following error window.

*)

//Version 0.00.06
//Cannon Melville
 FUNCTION AMC_StopMode
VAR_INPUT

	//If the AMC is commanded to stop.  There will be no ramp.
	bNo_Ramp_Stop				: BOOL := FALSE;  	
	
	
	//If the position error is larger then the following error window. 
	//Then the AMC will call a stop command. 
	bFollowing_Error_Stop		: BOOL := FALSE;  	
	
	
	//Max error before the AMC will cause the system to stop. If the Following_Error_Stop mode is true.
	diFollowing_Error_Window	: DINT ;
			
END_VAR

VAR_OUTPUT 
	
END_VAR

VAR
	myStopMode				: SINT;
END_VAR

(*	 
	Editing the code in this function may result in limited support. 	 
*)

(*Notes
	The code below uses fuctions to read and write to the drive.  The fuction format is shown below.
	WriteUserParameterUINT(Slot ,Menu	,Parameter, value );
	Value := ReadUserParameterDINT(Slot  ,Menu	,Parameter );
*)
	

